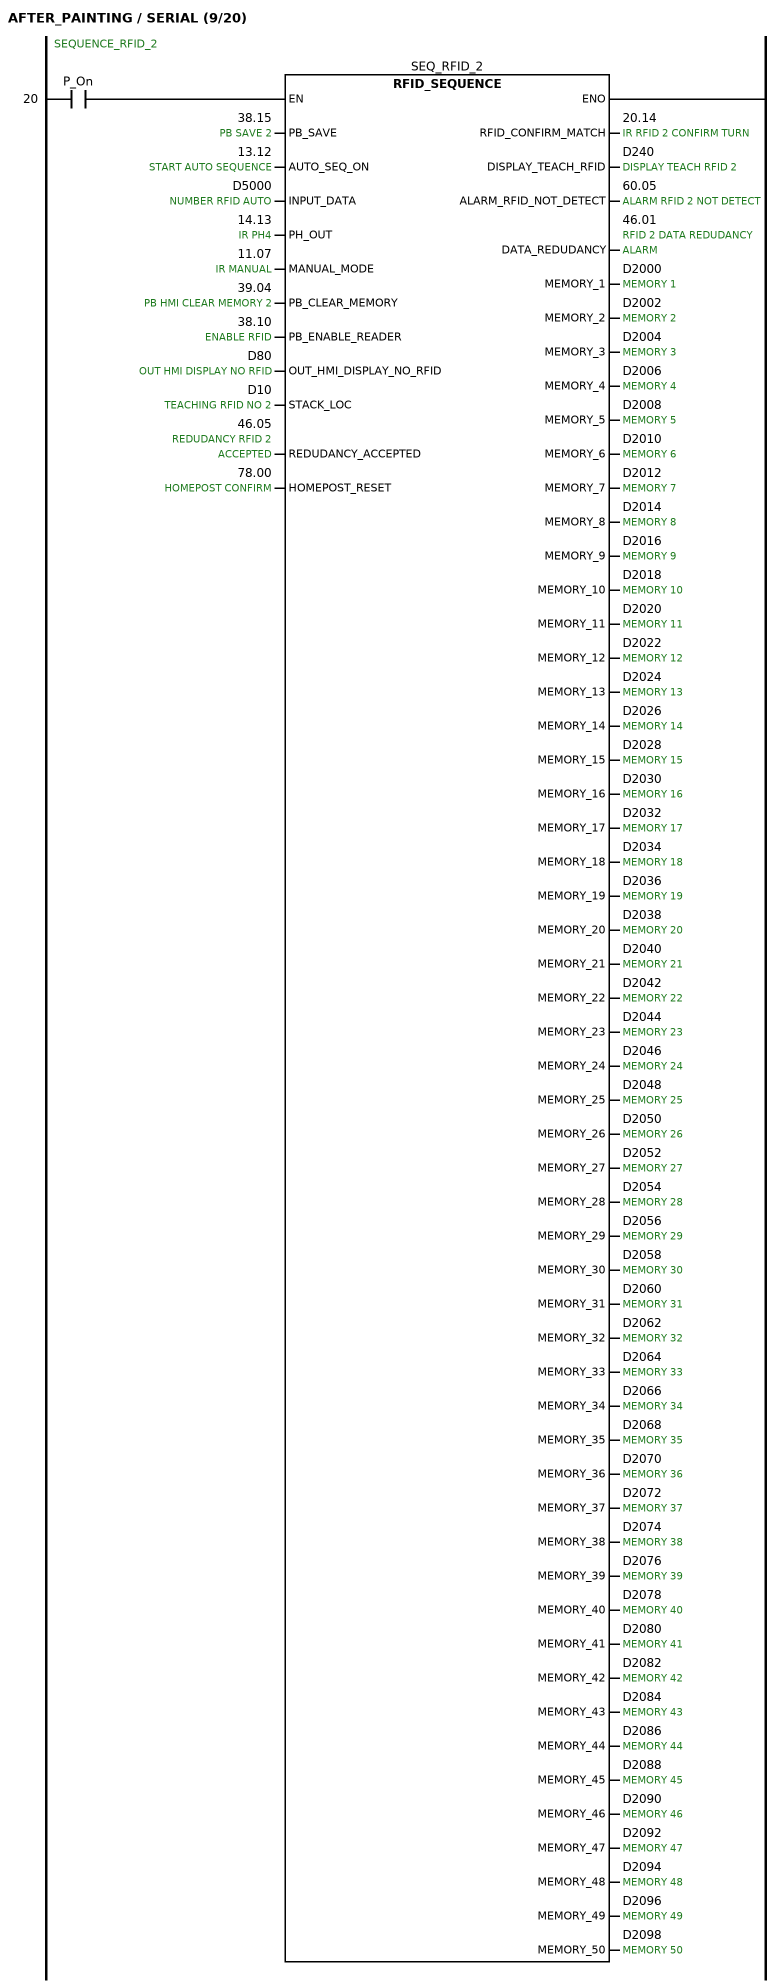
; [picture p72: AFTER_PAINTING / SERIAL, rungs 20-20]
; rung 20: SEQUENCE_RFID_2
LD P_On
CALL SEQ_RFID_2 : RFID_SEQUENCE (PB_SAVE := 38.15, AUTO_SEQ_ON := 13.12, INPUT_DATA := D5000, PH_OUT := 14.13, MANUAL_MODE := 11.07, PB_CLEAR_MEMORY := 39.04, PB_ENABLE_READER := 38.10, OUT_HMI_DISPLAY_NO_RFID := D80, STACK_LOC := D10, REDUDANCY_ACCEPTED := 46.05, HOMEPOST_RESET := 78.00, RFID_CONFIRM_MATCH => 20.14, DISPLAY_TEACH_RFID => D240, ALARM_RFID_NOT_DETECT => 60.05, DATA_REDUDANCY => 46.01, MEMORY_1 => D2000, MEMORY_2 => D2002, MEMORY_3 => D2004, MEMORY_4 => D2006, MEMORY_5 => D2008, MEMORY_6 => D2010, MEMORY_7 => D2012, MEMORY_8 => D2014, MEMORY_9 => D2016, MEMORY_10 => D2018, MEMORY_11 => D2020, MEMORY_12 => D2022, MEMORY_13 => D2024, MEMORY_14 => D2026, MEMORY_15 => D2028, MEMORY_16 => D2030, MEMORY_17 => D2032, MEMORY_18 => D2034, MEMORY_19 => D2036, MEMORY_20 => D2038, MEMORY_21 => D2040, MEMORY_22 => D2042, MEMORY_23 => D2044, MEMORY_24 => D2046, MEMORY_25 => D2048, MEMORY_26 => D2050, MEMORY_27 => D2052, MEMORY_28 => D2054, MEMORY_29 => D2056, MEMORY_30 => D2058, MEMORY_31 => D2060, MEMORY_32 => D2062, MEMORY_33 => D2064, MEMORY_34 => D2066, MEMORY_35 => D2068, MEMORY_36 => D2070, MEMORY_37 => D2072, MEMORY_38 => D2074, MEMORY_39 => D2076, MEMORY_40 => D2078, MEMORY_41 => D2080, MEMORY_42 => D2082, MEMORY_43 => D2084, MEMORY_44 => D2086, MEMORY_45 => D2088, MEMORY_46 => D2090, MEMORY_47 => D2092, MEMORY_48 => D2094, MEMORY_49 => D2096, MEMORY_50 => D2098)  ; PB SAVE 2, START AUTO SEQUENCE, NUMBER RFID AUTO, IR PH4, IR MANUAL, PB HMI CLEAR MEMORY 2, ENABLE RFID, OUT HMI DISPLAY NO RFID, TEACHING RFID NO 2, REDUDANCY RFID 2 ACCEPTED, HOMEPOST CONFIRM, IR RFID 2 CONFIRM TURN, DISPLAY TEACH RFID 2, ALARM RFID 2 NOT DETECT, RFID 2 DATA REDUDANCY ALARM, MEMORY 1, MEMORY 2, MEMORY 3, MEMORY 4, MEMORY 5, MEMORY 6, MEMORY 7, MEMORY 8, MEMORY 9, MEMORY 10, MEMORY 11, MEMORY 12, MEMORY 13, MEMORY 14, MEMORY 15, MEMORY 16, MEMORY 17, MEMORY 18, MEMORY 19, MEMORY 20, MEMORY 21, MEMORY 22, MEMORY 23, MEMORY 24, MEMORY 25, MEMORY 26, MEMORY 27, MEMORY 28, MEMORY 29, MEMORY 30, MEMORY 31, MEMORY 32, MEMORY 33, MEMORY 34, MEMORY 35, MEMORY 36, MEMORY 37, MEMORY 38, MEMORY 39, MEMORY 40, MEMORY 41, MEMORY 42, MEMORY 43, MEMORY 44, MEMORY 45, MEMORY 46, MEMORY 47, MEMORY 48, MEMORY 49, MEMORY 50

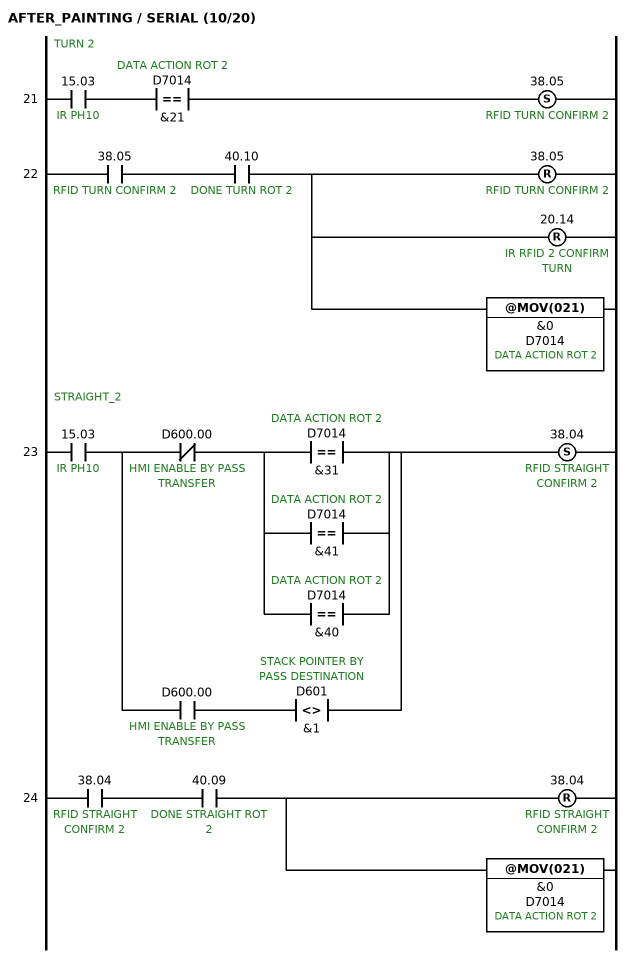
; rung 21: TURN 2
LD 15.03  ; IR PH10
AND=(300) D7014 &21  ; DATA ACTION ROT 2
SET 38.05  ; RFID TURN CONFIRM 2
; rung 22
LD 38.05  ; RFID TURN CONFIRM 2
AND 40.10  ; DONE TURN ROT 2
RSET 38.05  ; RFID TURN CONFIRM 2
RSET 20.14  ; IR RFID 2 CONFIRM TURN
@MOV(021) &0 D7014  ; DATA ACTION ROT 2
; rung 23: STRAIGHT_2
LD 15.03  ; IR PH10
LDNOT D600.00  ; HMI ENABLE BY PASS TRANSFER
LD=(300) D7014 &31  ; DATA ACTION ROT 2
OR=(300) D7014 &41  ; DATA ACTION ROT 2
OR=(300) D7014 &40  ; DATA ACTION ROT 2
ANDLD
LD D600.00  ; HMI ENABLE BY PASS TRANSFER
AND<>(305) D601 &1  ; STACK POINTER BY PASS DESTINATION
ORLD
ANDLD
SET 38.04  ; RFID STRAIGHT CONFIRM 2
; rung 24
LD 38.04  ; RFID STRAIGHT CONFIRM 2
AND 40.09  ; DONE STRAIGHT ROT 2
RSET 38.04  ; RFID STRAIGHT CONFIRM 2
@MOV(021) &0 D7014  ; DATA ACTION ROT 2

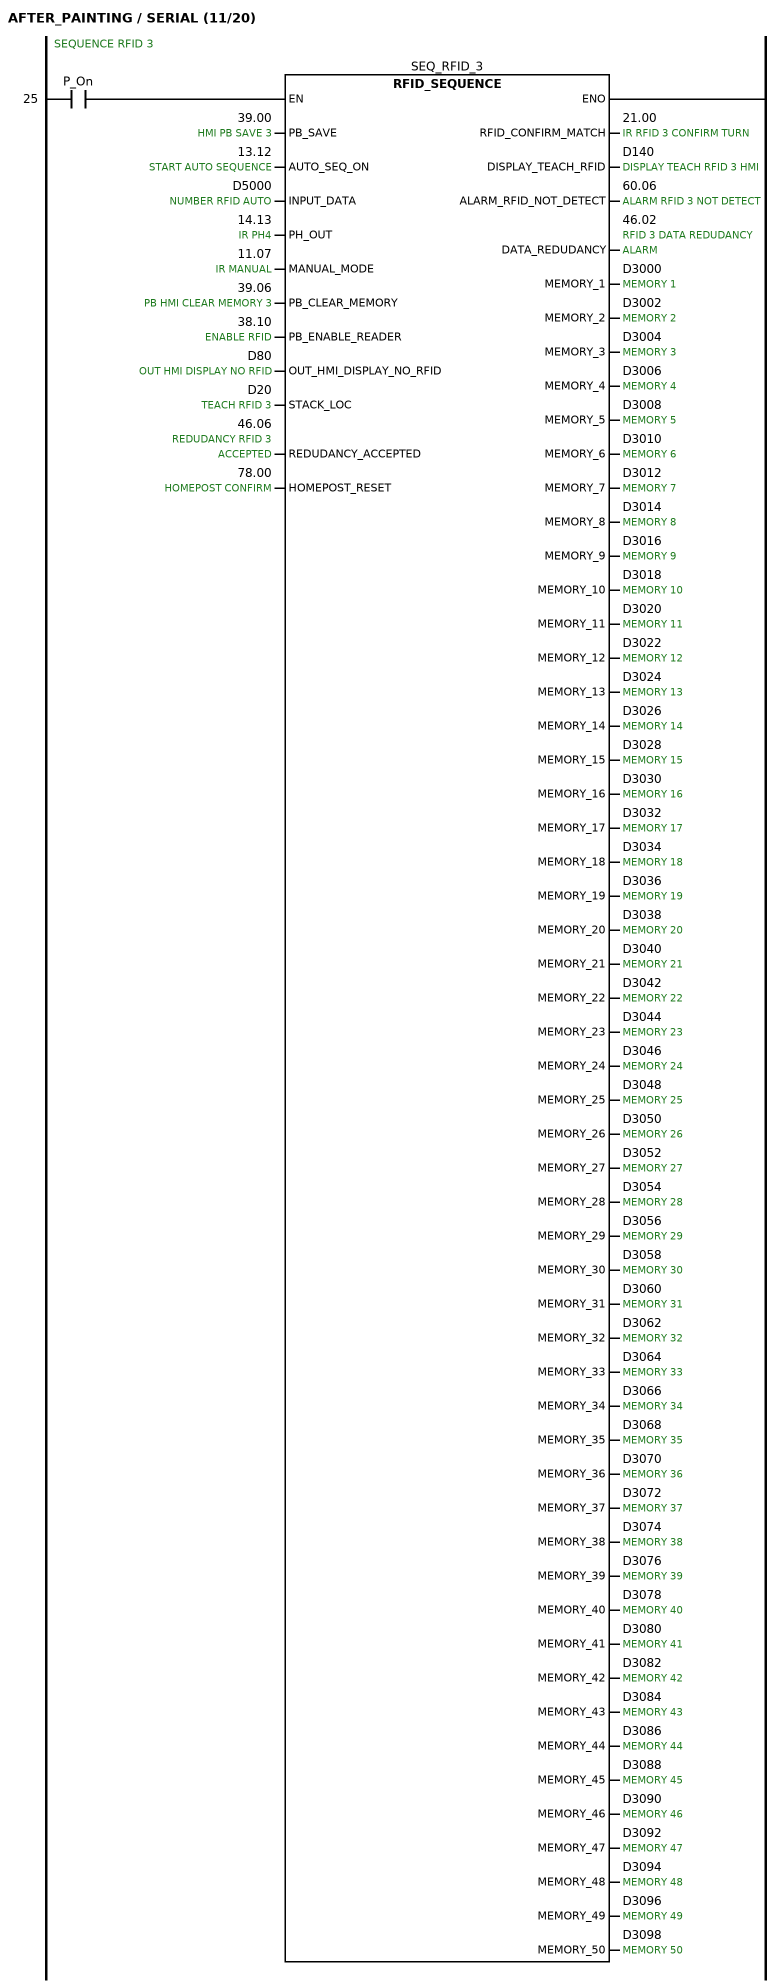
; rung 25: SEQUENCE RFID 3
LD P_On
CALL SEQ_RFID_3 : RFID_SEQUENCE (PB_SAVE := 39.00, AUTO_SEQ_ON := 13.12, INPUT_DATA := D5000, PH_OUT := 14.13, MANUAL_MODE := 11.07, PB_CLEAR_MEMORY := 39.06, PB_ENABLE_READER := 38.10, OUT_HMI_DISPLAY_NO_RFID := D80, STACK_LOC := D20, REDUDANCY_ACCEPTED := 46.06, HOMEPOST_RESET := 78.00, RFID_CONFIRM_MATCH => 21.00, DISPLAY_TEACH_RFID => D140, ALARM_RFID_NOT_DETECT => 60.06, DATA_REDUDANCY => 46.02, MEMORY_1 => D3000, MEMORY_2 => D3002, MEMORY_3 => D3004, MEMORY_4 => D3006, MEMORY_5 => D3008, MEMORY_6 => D3010, MEMORY_7 => D3012, MEMORY_8 => D3014, MEMORY_9 => D3016, MEMORY_10 => D3018, MEMORY_11 => D3020, MEMORY_12 => D3022, MEMORY_13 => D3024, MEMORY_14 => D3026, MEMORY_15 => D3028, MEMORY_16 => D3030, MEMORY_17 => D3032, MEMORY_18 => D3034, MEMORY_19 => D3036, MEMORY_20 => D3038, MEMORY_21 => D3040, MEMORY_22 => D3042, MEMORY_23 => D3044, MEMORY_24 => D3046, MEMORY_25 => D3048, MEMORY_26 => D3050, MEMORY_27 => D3052, MEMORY_28 => D3054, MEMORY_29 => D3056, MEMORY_30 => D3058, MEMORY_31 => D3060, MEMORY_32 => D3062, MEMORY_33 => D3064, MEMORY_34 => D3066, MEMORY_35 => D3068, MEMORY_36 => D3070, MEMORY_37 => D3072, MEMORY_38 => D3074, MEMORY_39 => D3076, MEMORY_40 => D3078, MEMORY_41 => D3080, MEMORY_42 => D3082, MEMORY_43 => D3084, MEMORY_44 => D3086, MEMORY_45 => D3088, MEMORY_46 => D3090, MEMORY_47 => D3092, MEMORY_48 => D3094, MEMORY_49 => D3096, MEMORY_50 => D3098)  ; HMI PB SAVE 3, START AUTO SEQUENCE, NUMBER RFID AUTO, IR PH4, IR MANUAL, PB HMI CLEAR MEMORY 3, ENABLE RFID, OUT HMI DISPLAY NO RFID, TEACH RFID 3, REDUDANCY RFID 3 ACCEPTED, HOMEPOST CONFIRM, IR RFID 3 CONFIRM TURN, DISPLAY TEACH RFID 3 HMI, ALARM RFID 3 NOT DETECT, RFID 3 DATA REDUDANCY ALARM, MEMORY 1, MEMORY 2, MEMORY 3, MEMORY 4, MEMORY 5, MEMORY 6, MEMORY 7, MEMORY 8, MEMORY 9, MEMORY 10, MEMORY 11, MEMORY 12, MEMORY 13, MEMORY 14, MEMORY 15, MEMORY 16, MEMORY 17, MEMORY 18, MEMORY 19, MEMORY 20, MEMORY 21, MEMORY 22, MEMORY 23, MEMORY 24, MEMORY 25, MEMORY 26, MEMORY 27, MEMORY 28, MEMORY 29, MEMORY 30, MEMORY 31, MEMORY 32, MEMORY 33, MEMORY 34, MEMORY 35, MEMORY 36, MEMORY 37, MEMORY 38, MEMORY 39, MEMORY 40, MEMORY 41, MEMORY 42, MEMORY 43, MEMORY 44, MEMORY 45, MEMORY 46, MEMORY 47, MEMORY 48, MEMORY 49, MEMORY 50

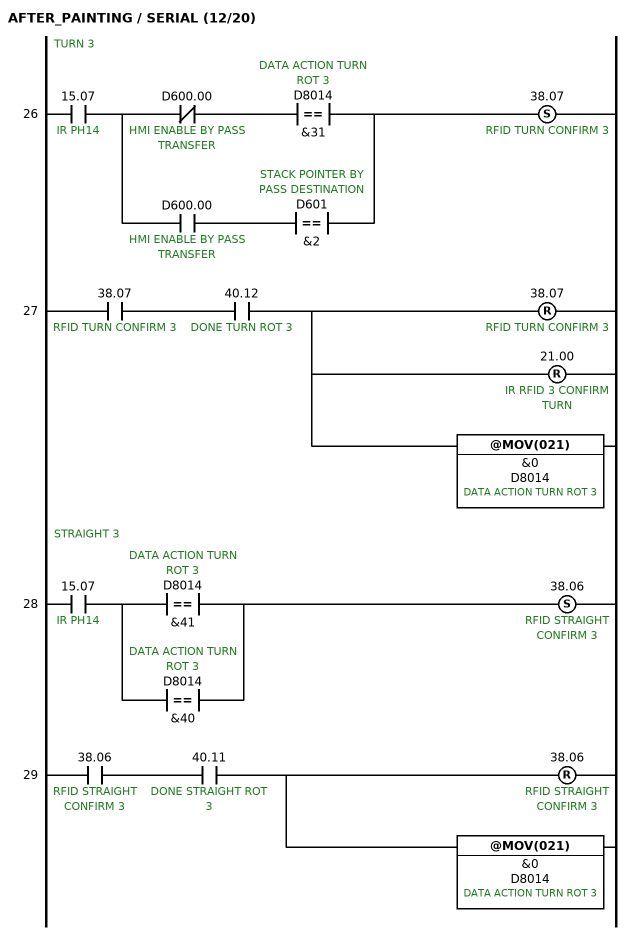
; rung 26: TURN 3
LD 15.07  ; IR PH14
LDNOT D600.00  ; HMI ENABLE BY PASS TRANSFER
AND=(300) D8014 &31  ; DATA ACTION TURN ROT 3
LD D600.00  ; HMI ENABLE BY PASS TRANSFER
AND=(300) D601 &2  ; STACK POINTER BY PASS DESTINATION
ORLD
ANDLD
SET 38.07  ; RFID TURN CONFIRM 3
; rung 27
LD 38.07  ; RFID TURN CONFIRM 3
AND 40.12  ; DONE TURN ROT 3
RSET 38.07  ; RFID TURN CONFIRM 3
RSET 21.00  ; IR RFID 3 CONFIRM TURN
@MOV(021) &0 D8014  ; DATA ACTION TURN ROT 3
; rung 28: STRAIGHT 3
LD 15.07  ; IR PH14
LD=(300) D8014 &41  ; DATA ACTION TURN ROT 3
OR=(300) D8014 &40  ; DATA ACTION TURN ROT 3
ANDLD
SET 38.06  ; RFID STRAIGHT CONFIRM 3
; rung 29
LD 38.06  ; RFID STRAIGHT CONFIRM 3
AND 40.11  ; DONE STRAIGHT ROT 3
RSET 38.06  ; RFID STRAIGHT CONFIRM 3
@MOV(021) &0 D8014  ; DATA ACTION TURN ROT 3

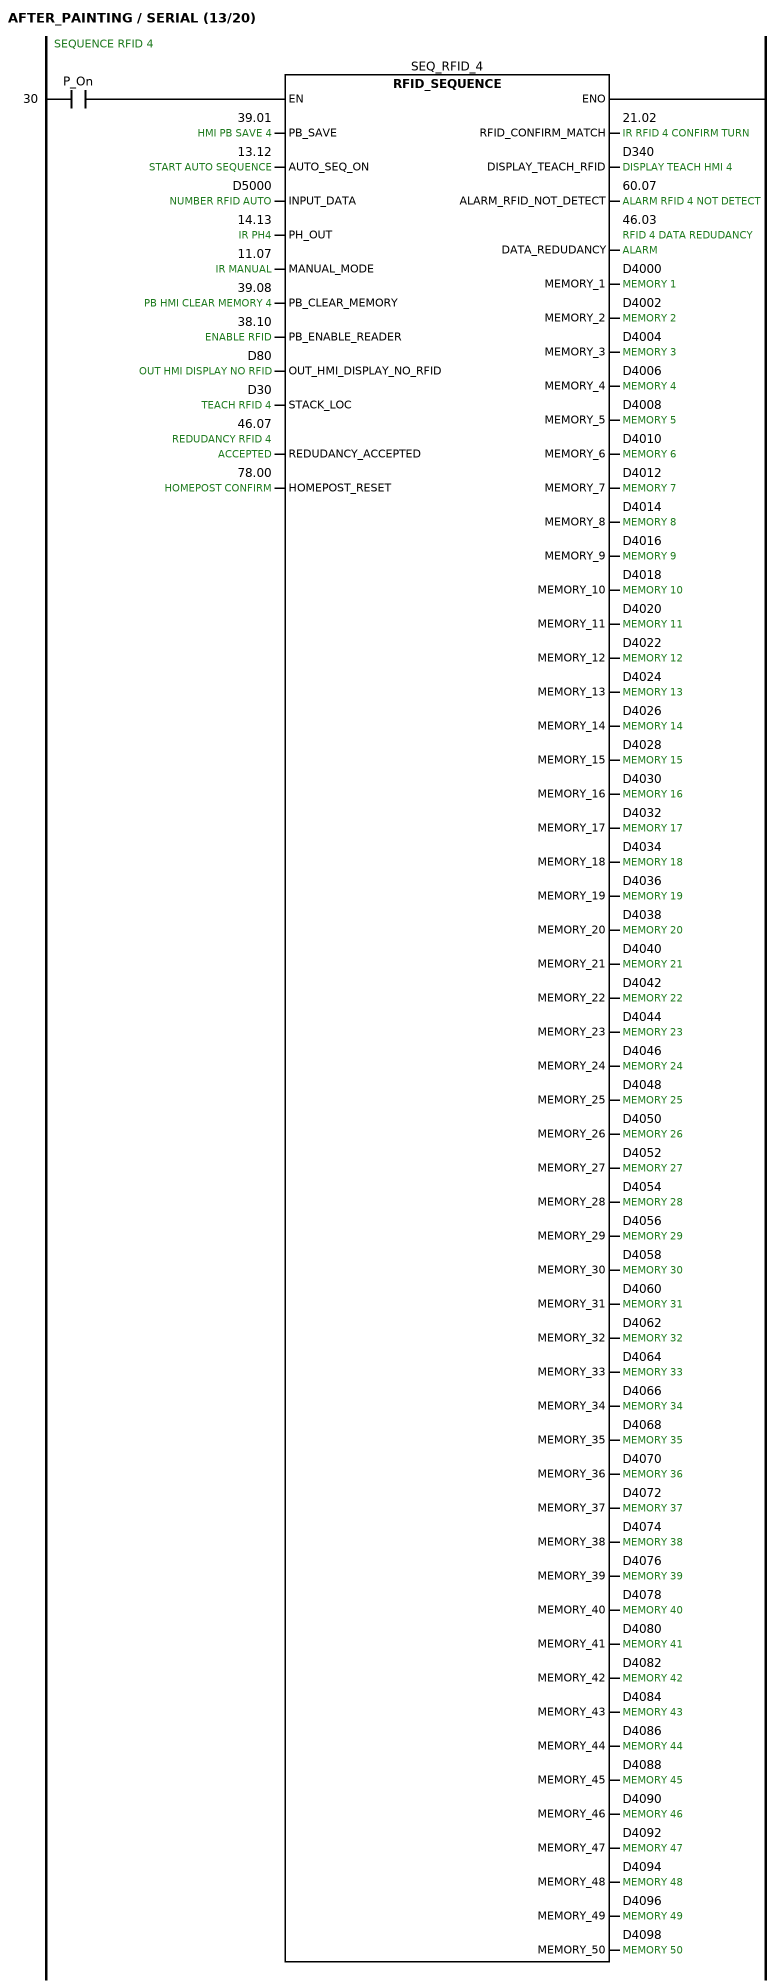
; rung 30: SEQUENCE RFID 4
LD P_On
CALL SEQ_RFID_4 : RFID_SEQUENCE (PB_SAVE := 39.01, AUTO_SEQ_ON := 13.12, INPUT_DATA := D5000, PH_OUT := 14.13, MANUAL_MODE := 11.07, PB_CLEAR_MEMORY := 39.08, PB_ENABLE_READER := 38.10, OUT_HMI_DISPLAY_NO_RFID := D80, STACK_LOC := D30, REDUDANCY_ACCEPTED := 46.07, HOMEPOST_RESET := 78.00, RFID_CONFIRM_MATCH => 21.02, DISPLAY_TEACH_RFID => D340, ALARM_RFID_NOT_DETECT => 60.07, DATA_REDUDANCY => 46.03, MEMORY_1 => D4000, MEMORY_2 => D4002, MEMORY_3 => D4004, MEMORY_4 => D4006, MEMORY_5 => D4008, MEMORY_6 => D4010, MEMORY_7 => D4012, MEMORY_8 => D4014, MEMORY_9 => D4016, MEMORY_10 => D4018, MEMORY_11 => D4020, MEMORY_12 => D4022, MEMORY_13 => D4024, MEMORY_14 => D4026, MEMORY_15 => D4028, MEMORY_16 => D4030, MEMORY_17 => D4032, MEMORY_18 => D4034, MEMORY_19 => D4036, MEMORY_20 => D4038, MEMORY_21 => D4040, MEMORY_22 => D4042, MEMORY_23 => D4044, MEMORY_24 => D4046, MEMORY_25 => D4048, MEMORY_26 => D4050, MEMORY_27 => D4052, MEMORY_28 => D4054, MEMORY_29 => D4056, MEMORY_30 => D4058, MEMORY_31 => D4060, MEMORY_32 => D4062, MEMORY_33 => D4064, MEMORY_34 => D4066, MEMORY_35 => D4068, MEMORY_36 => D4070, MEMORY_37 => D4072, MEMORY_38 => D4074, MEMORY_39 => D4076, MEMORY_40 => D4078, MEMORY_41 => D4080, MEMORY_42 => D4082, MEMORY_43 => D4084, MEMORY_44 => D4086, MEMORY_45 => D4088, MEMORY_46 => D4090, MEMORY_47 => D4092, MEMORY_48 => D4094, MEMORY_49 => D4096, MEMORY_50 => D4098)  ; HMI PB SAVE 4, START AUTO SEQUENCE, NUMBER RFID AUTO, IR PH4, IR MANUAL, PB HMI CLEAR MEMORY 4, ENABLE RFID, OUT HMI DISPLAY NO RFID, TEACH RFID 4, REDUDANCY RFID 4 ACCEPTED, HOMEPOST CONFIRM, IR RFID 4 CONFIRM TURN, DISPLAY TEACH HMI 4, ALARM RFID 4 NOT DETECT, RFID 4 DATA REDUDANCY ALARM, MEMORY 1, MEMORY 2, MEMORY 3, MEMORY 4, MEMORY 5, MEMORY 6, MEMORY 7, MEMORY 8, MEMORY 9, MEMORY 10, MEMORY 11, MEMORY 12, MEMORY 13, MEMORY 14, MEMORY 15, MEMORY 16, MEMORY 17, MEMORY 18, MEMORY 19, MEMORY 20, MEMORY 21, MEMORY 22, MEMORY 23, MEMORY 24, MEMORY 25, MEMORY 26, MEMORY 27, MEMORY 28, MEMORY 29, MEMORY 30, MEMORY 31, MEMORY 32, MEMORY 33, MEMORY 34, MEMORY 35, MEMORY 36, MEMORY 37, MEMORY 38, MEMORY 39, MEMORY 40, MEMORY 41, MEMORY 42, MEMORY 43, MEMORY 44, MEMORY 45, MEMORY 46, MEMORY 47, MEMORY 48, MEMORY 49, MEMORY 50

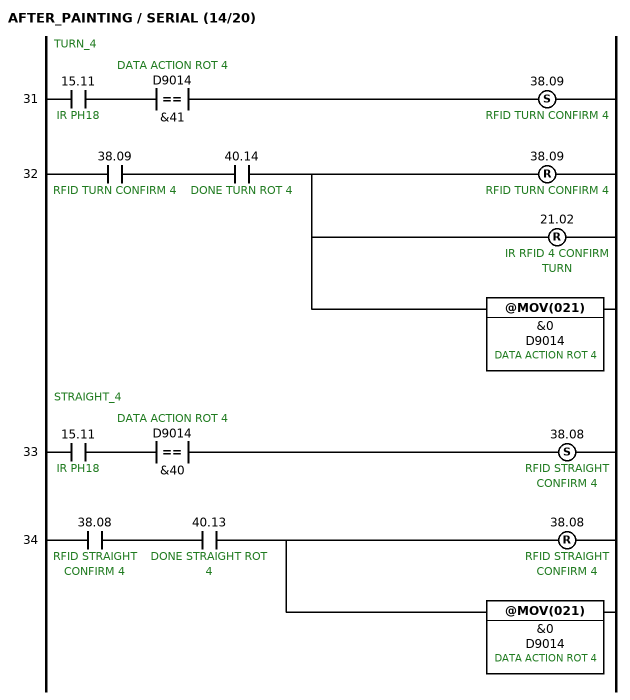
; rung 31: TURN_4
LD 15.11  ; IR PH18
AND=(300) D9014 &41  ; DATA ACTION ROT 4
SET 38.09  ; RFID TURN CONFIRM 4
; rung 32
LD 38.09  ; RFID TURN CONFIRM 4
AND 40.14  ; DONE TURN ROT 4
RSET 38.09  ; RFID TURN CONFIRM 4
RSET 21.02  ; IR RFID 4 CONFIRM TURN
@MOV(021) &0 D9014  ; DATA ACTION ROT 4
; rung 33: STRAIGHT_4
LD 15.11  ; IR PH18
AND=(300) D9014 &40  ; DATA ACTION ROT 4
SET 38.08  ; RFID STRAIGHT CONFIRM 4
; rung 34
LD 38.08  ; RFID STRAIGHT CONFIRM 4
AND 40.13  ; DONE STRAIGHT ROT 4
RSET 38.08  ; RFID STRAIGHT CONFIRM 4
@MOV(021) &0 D9014  ; DATA ACTION ROT 4

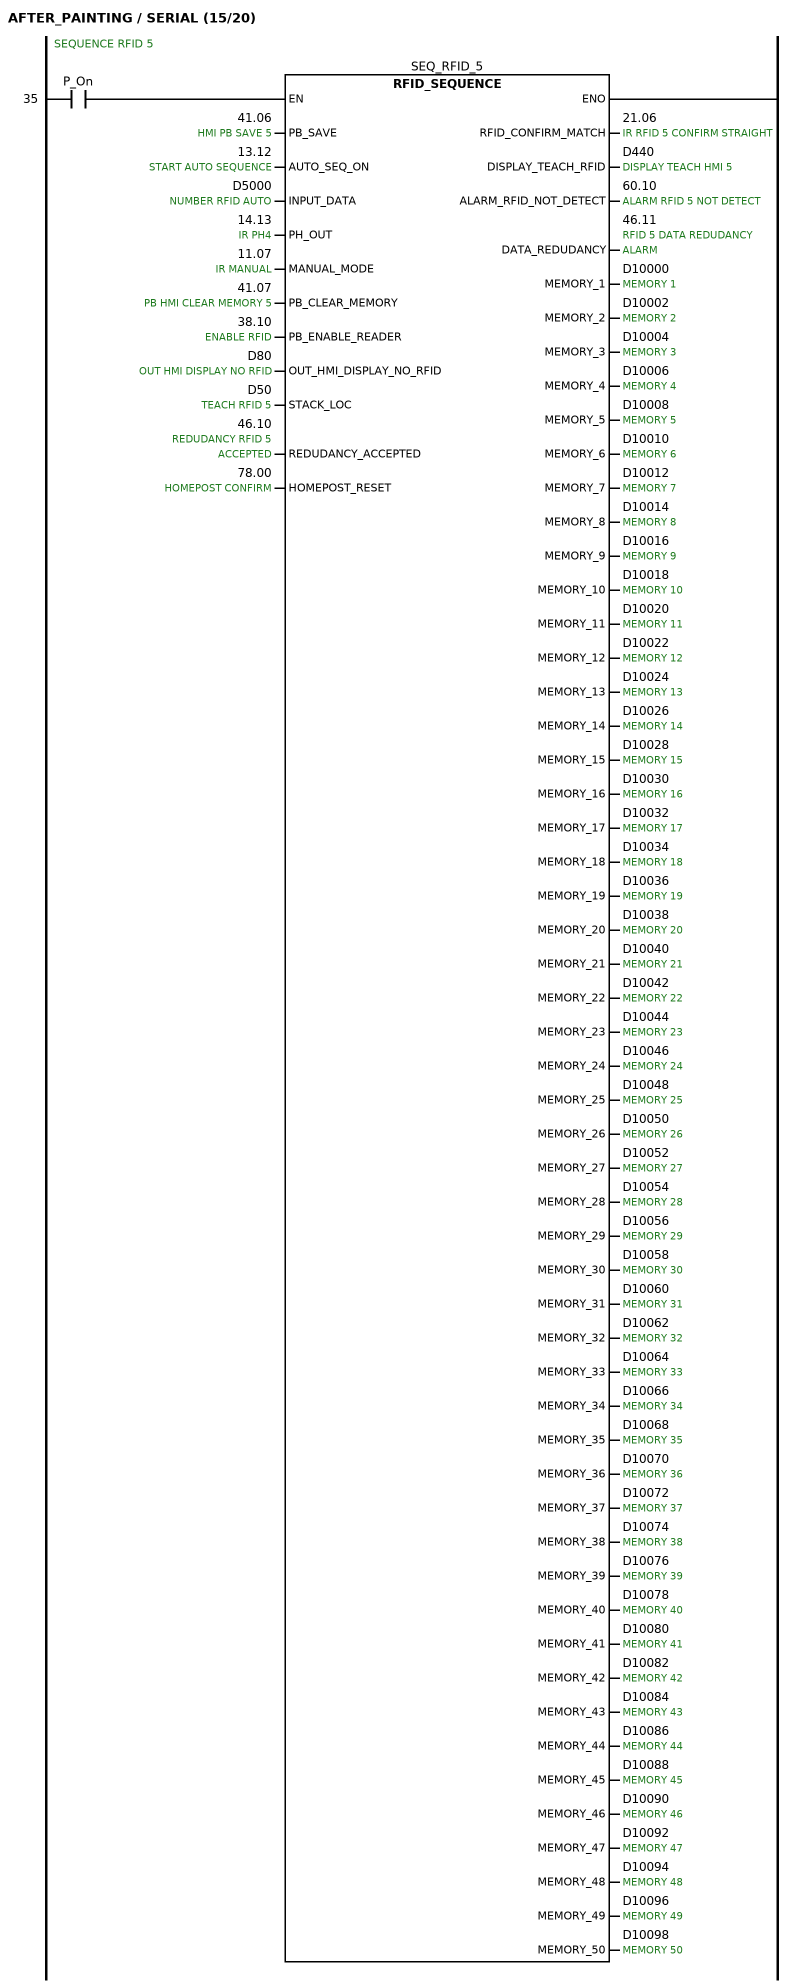
; rung 35: SEQUENCE RFID 5
LD P_On
CALL SEQ_RFID_5 : RFID_SEQUENCE (PB_SAVE := 41.06, AUTO_SEQ_ON := 13.12, INPUT_DATA := D5000, PH_OUT := 14.13, MANUAL_MODE := 11.07, PB_CLEAR_MEMORY := 41.07, PB_ENABLE_READER := 38.10, OUT_HMI_DISPLAY_NO_RFID := D80, STACK_LOC := D50, REDUDANCY_ACCEPTED := 46.10, HOMEPOST_RESET := 78.00, RFID_CONFIRM_MATCH => 21.06, DISPLAY_TEACH_RFID => D440, ALARM_RFID_NOT_DETECT => 60.10, DATA_REDUDANCY => 46.11, MEMORY_1 => D10000, MEMORY_2 => D10002, MEMORY_3 => D10004, MEMORY_4 => D10006, MEMORY_5 => D10008, MEMORY_6 => D10010, MEMORY_7 => D10012, MEMORY_8 => D10014, MEMORY_9 => D10016, MEMORY_10 => D10018, MEMORY_11 => D10020, MEMORY_12 => D10022, MEMORY_13 => D10024, MEMORY_14 => D10026, MEMORY_15 => D10028, MEMORY_16 => D10030, MEMORY_17 => D10032, MEMORY_18 => D10034, MEMORY_19 => D10036, MEMORY_20 => D10038, MEMORY_21 => D10040, MEMORY_22 => D10042, MEMORY_23 => D10044, MEMORY_24 => D10046, MEMORY_25 => D10048, MEMORY_26 => D10050, MEMORY_27 => D10052, MEMORY_28 => D10054, MEMORY_29 => D10056, MEMORY_30 => D10058, MEMORY_31 => D10060, MEMORY_32 => D10062, MEMORY_33 => D10064, MEMORY_34 => D10066, MEMORY_35 => D10068, MEMORY_36 => D10070, MEMORY_37 => D10072, MEMORY_38 => D10074, MEMORY_39 => D10076, MEMORY_40 => D10078, MEMORY_41 => D10080, MEMORY_42 => D10082, MEMORY_43 => D10084, MEMORY_44 => D10086, MEMORY_45 => D10088, MEMORY_46 => D10090, MEMORY_47 => D10092, MEMORY_48 => D10094, MEMORY_49 => D10096, MEMORY_50 => D10098)  ; HMI PB SAVE 5, START AUTO SEQUENCE, NUMBER RFID AUTO, IR PH4, IR MANUAL, PB HMI CLEAR MEMORY 5, ENABLE RFID, OUT HMI DISPLAY NO RFID, TEACH RFID 5, REDUDANCY RFID 5 ACCEPTED, HOMEPOST CONFIRM, IR RFID 5 CONFIRM STRAIGHT, DISPLAY TEACH HMI 5, ALARM RFID 5 NOT DETECT, RFID 5 DATA REDUDANCY ALARM, MEMORY 1, MEMORY 2, MEMORY 3, MEMORY 4, MEMORY 5, MEMORY 6, MEMORY 7, MEMORY 8, MEMORY 9, MEMORY 10, MEMORY 11, MEMORY 12, MEMORY 13, MEMORY 14, MEMORY 15, MEMORY 16, MEMORY 17, MEMORY 18, MEMORY 19, MEMORY 20, MEMORY 21, MEMORY 22, MEMORY 23, MEMORY 24, MEMORY 25, MEMORY 26, MEMORY 27, MEMORY 28, MEMORY 29, MEMORY 30, MEMORY 31, MEMORY 32, MEMORY 33, MEMORY 34, MEMORY 35, MEMORY 36, MEMORY 37, MEMORY 38, MEMORY 39, MEMORY 40, MEMORY 41, MEMORY 42, MEMORY 43, MEMORY 44, MEMORY 45, MEMORY 46, MEMORY 47, MEMORY 48, MEMORY 49, MEMORY 50

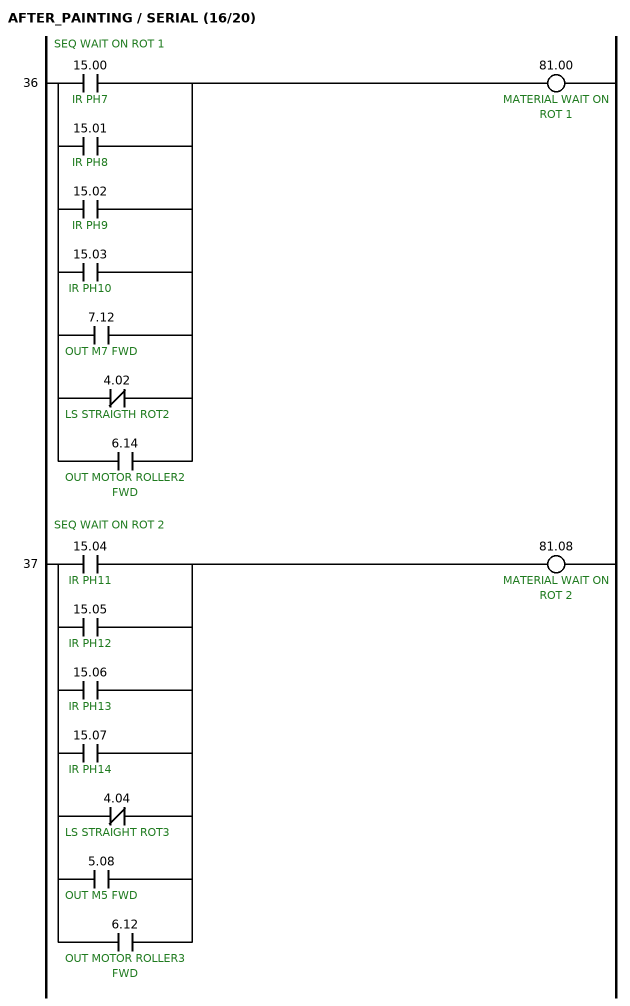
; rung 36: SEQ WAIT ON ROT 1
LD 15.00  ; IR PH7
OR 15.01  ; IR PH8
OR 15.02  ; IR PH9
OR 15.03  ; IR PH10
OR 7.12  ; OUT M7 FWD
ORNOT 4.02  ; LS STRAIGTH ROT2
OR 6.14  ; OUT MOTOR ROLLER2 FWD
OUT 81.00  ; MATERIAL WAIT ON ROT 1
; rung 37: SEQ WAIT ON ROT 2
LD 15.04  ; IR PH11
OR 15.05  ; IR PH12
OR 15.06  ; IR PH13
OR 15.07  ; IR PH14
ORNOT 4.04  ; LS STRAIGHT ROT3
OR 5.08  ; OUT M5 FWD
OR 6.12  ; OUT MOTOR ROLLER3 FWD
OUT 81.08  ; MATERIAL WAIT ON ROT 2

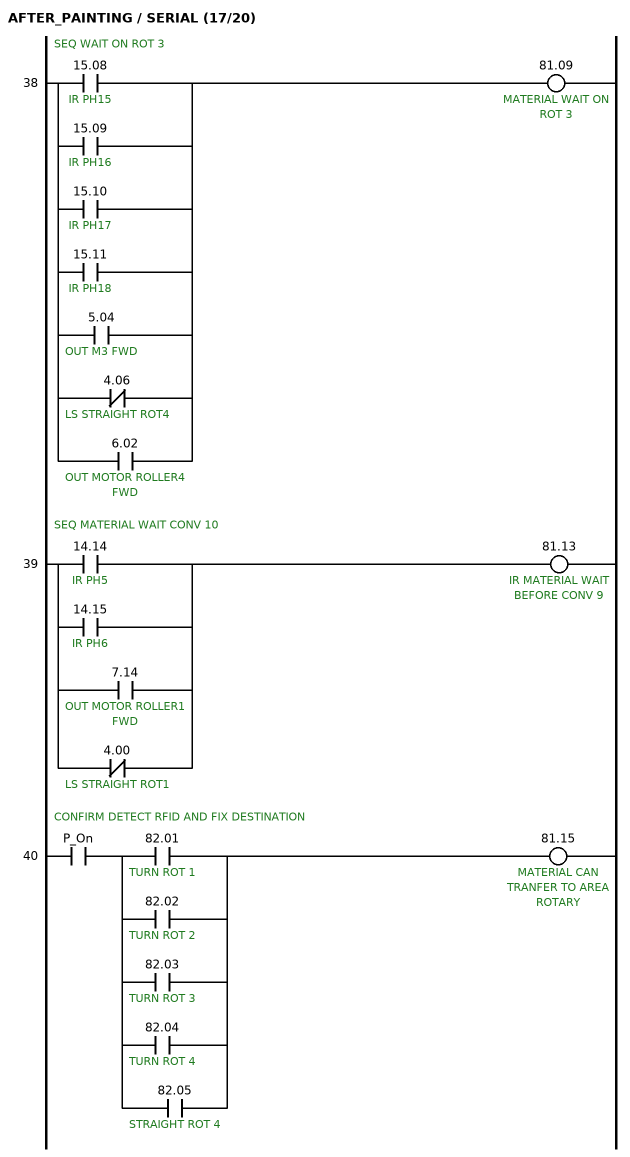
; rung 38: SEQ WAIT ON ROT 3
LD 15.08  ; IR PH15
OR 15.09  ; IR PH16
OR 15.10  ; IR PH17
OR 15.11  ; IR PH18
OR 5.04  ; OUT M3 FWD
ORNOT 4.06  ; LS STRAIGHT ROT4
OR 6.02  ; OUT MOTOR ROLLER4 FWD
OUT 81.09  ; MATERIAL WAIT ON ROT 3
; rung 39: SEQ MATERIAL WAIT CONV 10
LD 14.14  ; IR PH5
OR 14.15  ; IR PH6
OR 7.14  ; OUT MOTOR ROLLER1 FWD
ORNOT 4.00  ; LS STRAIGHT ROT1
OUT 81.13  ; IR MATERIAL WAIT BEFORE CONV 9
; rung 40: CONFIRM DETECT RFID AND FIX DESTINATION
LD P_On
LD 82.01  ; TURN ROT 1
OR 82.02  ; TURN ROT 2
OR 82.03  ; TURN ROT 3
OR 82.04  ; TURN ROT 4
OR 82.05  ; STRAIGHT ROT 4
ANDLD
OUT 81.15  ; MATERIAL CAN TRANFER TO AREA ROTARY

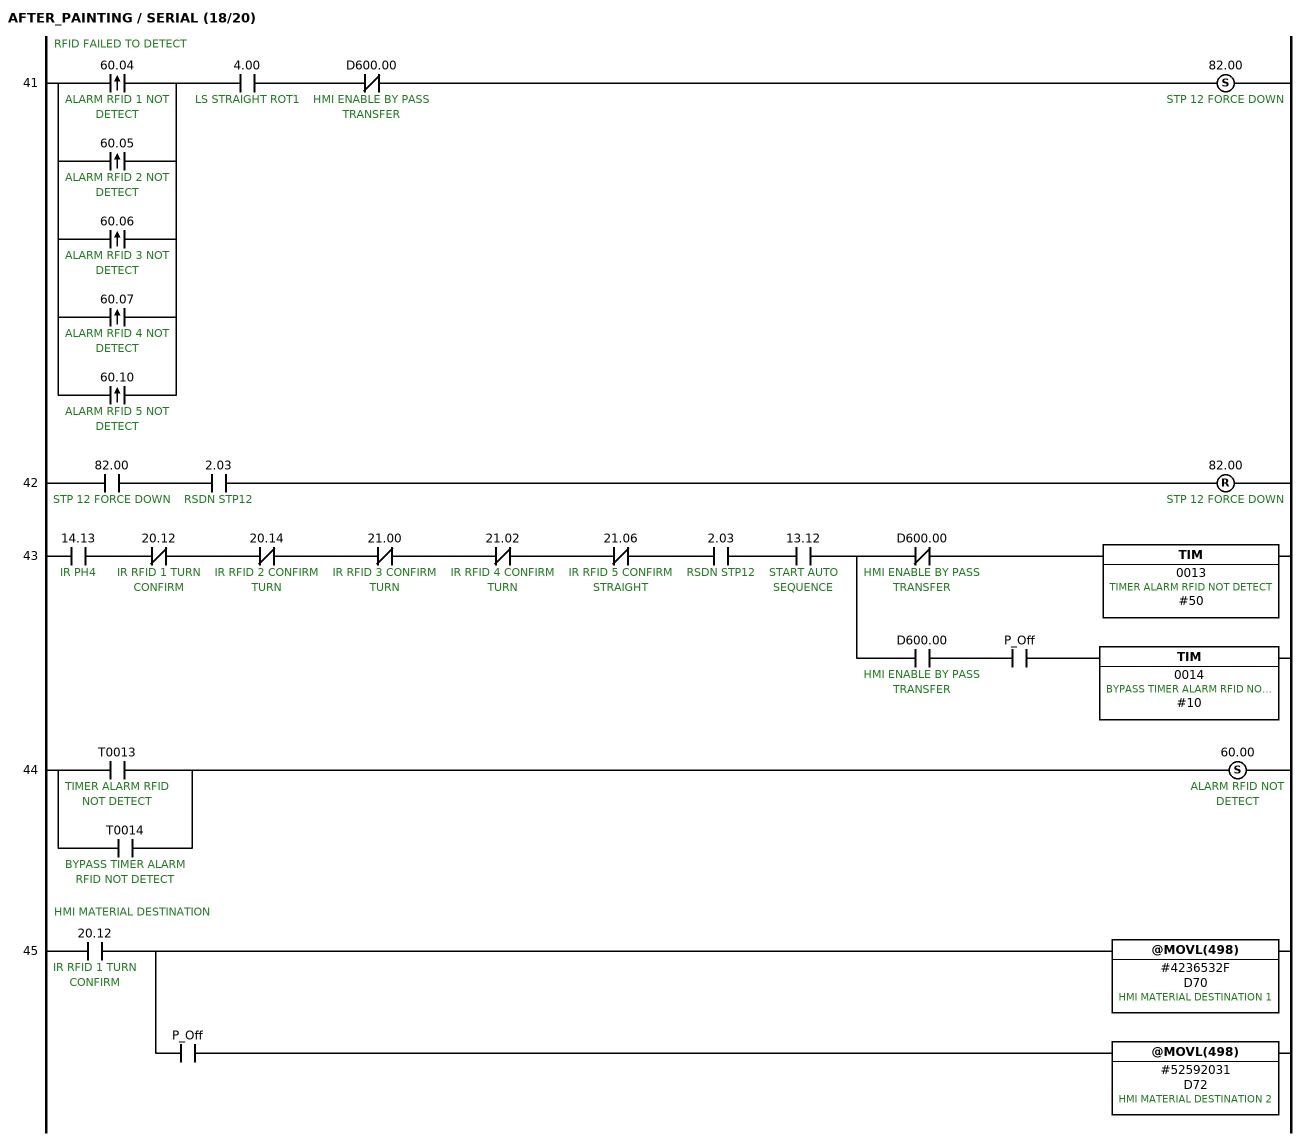
; rung 41: RFID FAILED TO DETECT
@LD 60.04  ; ALARM RFID 1 NOT DETECT
@OR 60.05  ; ALARM RFID 2 NOT DETECT
@OR 60.06  ; ALARM RFID 3 NOT DETECT
@OR 60.07  ; ALARM RFID 4 NOT DETECT
@OR 60.10  ; ALARM RFID 5 NOT DETECT
AND 4.00  ; LS STRAIGHT ROT1
ANDNOT D600.00  ; HMI ENABLE BY PASS TRANSFER
SET 82.00  ; STP 12 FORCE DOWN
; rung 42
LD 82.00  ; STP 12 FORCE DOWN
AND 2.03  ; RSDN STP12
RSET 82.00  ; STP 12 FORCE DOWN
; rung 43
LD 14.13  ; IR PH4
ANDNOT 20.12  ; IR RFID 1 TURN CONFIRM
ANDNOT 20.14  ; IR RFID 2 CONFIRM TURN
ANDNOT 21.00  ; IR RFID 3 CONFIRM TURN
ANDNOT 21.02  ; IR RFID 4 CONFIRM TURN
ANDNOT 21.06  ; IR RFID 5 CONFIRM STRAIGHT
AND 2.03  ; RSDN STP12
AND 13.12  ; START AUTO SEQUENCE
OUT TR0
ANDNOT D600.00  ; HMI ENABLE BY PASS TRANSFER
TIM 0013 #50  ; TIMER ALARM RFID NOT DETECT
LD TR0
AND D600.00  ; HMI ENABLE BY PASS TRANSFER
AND P_Off
TIM 0014 #10  ; BYPASS TIMER ALARM RFID NOT DETECT
; rung 44
LD T0013  ; TIMER ALARM RFID NOT DETECT
OR T0014  ; BYPASS TIMER ALARM RFID NOT DETECT
SET 60.00  ; ALARM RFID NOT DETECT
; rung 45: HMI MATERIAL DESTINATION
LD 20.12  ; IR RFID 1 TURN CONFIRM
@MOVL(498) #4236532F D70  ; HMI MATERIAL DESTINATION 1
AND P_Off
@MOVL(498) #52592031 D72  ; HMI MATERIAL DESTINATION 2

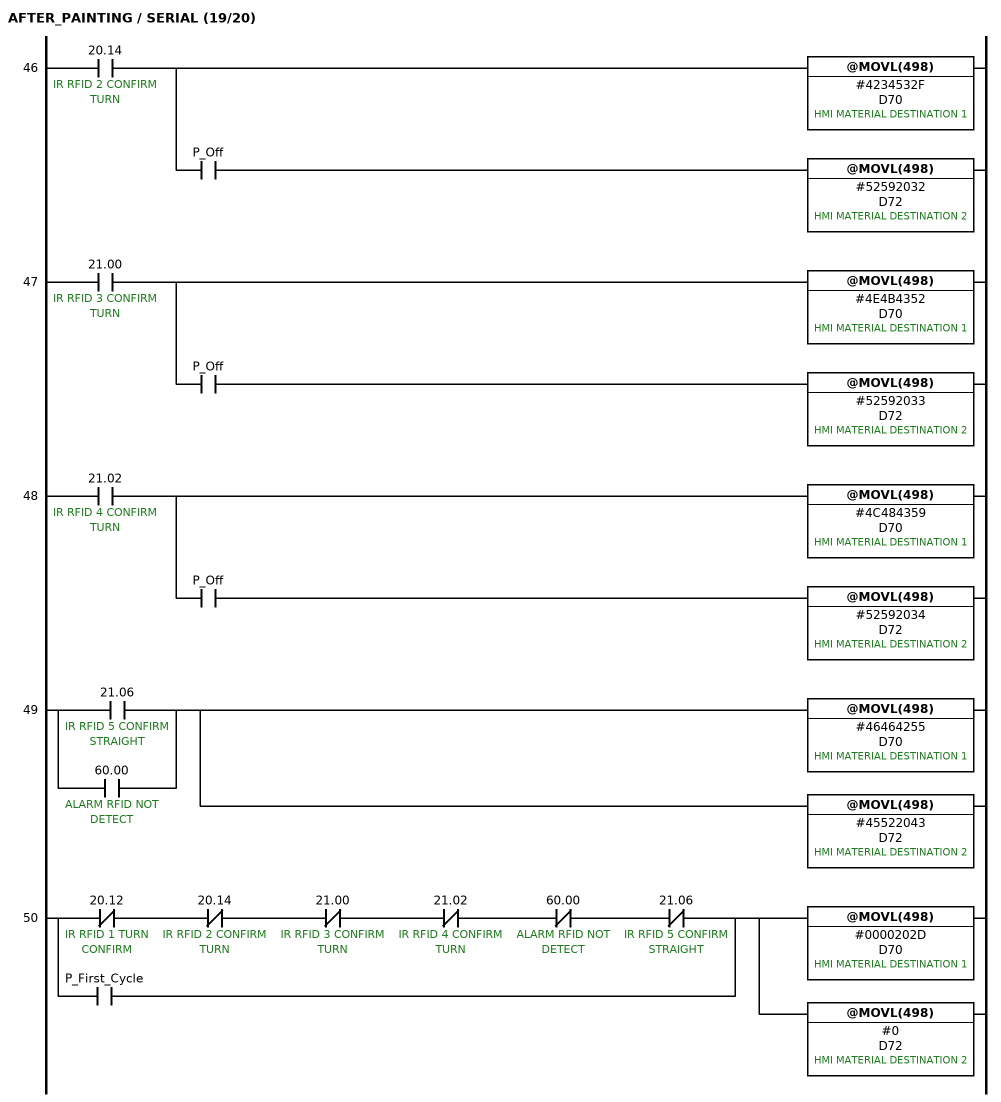
; rung 46
LD 20.14  ; IR RFID 2 CONFIRM TURN
@MOVL(498) #4234532F D70  ; HMI MATERIAL DESTINATION 1
AND P_Off
@MOVL(498) #52592032 D72  ; HMI MATERIAL DESTINATION 2
; rung 47
LD 21.00  ; IR RFID 3 CONFIRM TURN
@MOVL(498) #4E4B4352 D70  ; HMI MATERIAL DESTINATION 1
AND P_Off
@MOVL(498) #52592033 D72  ; HMI MATERIAL DESTINATION 2
; rung 48
LD 21.02  ; IR RFID 4 CONFIRM TURN
@MOVL(498) #4C484359 D70  ; HMI MATERIAL DESTINATION 1
AND P_Off
@MOVL(498) #52592034 D72  ; HMI MATERIAL DESTINATION 2
; rung 49
LD 21.06  ; IR RFID 5 CONFIRM STRAIGHT
OR 60.00  ; ALARM RFID NOT DETECT
@MOVL(498) #46464255 D70  ; HMI MATERIAL DESTINATION 1
@MOVL(498) #45522043 D72  ; HMI MATERIAL DESTINATION 2
; rung 50
LDNOT 20.12  ; IR RFID 1 TURN CONFIRM
ANDNOT 20.14  ; IR RFID 2 CONFIRM TURN
ANDNOT 21.00  ; IR RFID 3 CONFIRM TURN
ANDNOT 21.02  ; IR RFID 4 CONFIRM TURN
ANDNOT 60.00  ; ALARM RFID NOT DETECT
ANDNOT 21.06  ; IR RFID 5 CONFIRM STRAIGHT
OR P_First_Cycle
@MOVL(498) #0000202D D70  ; HMI MATERIAL DESTINATION 1
@MOVL(498) #0 D72  ; HMI MATERIAL DESTINATION 2

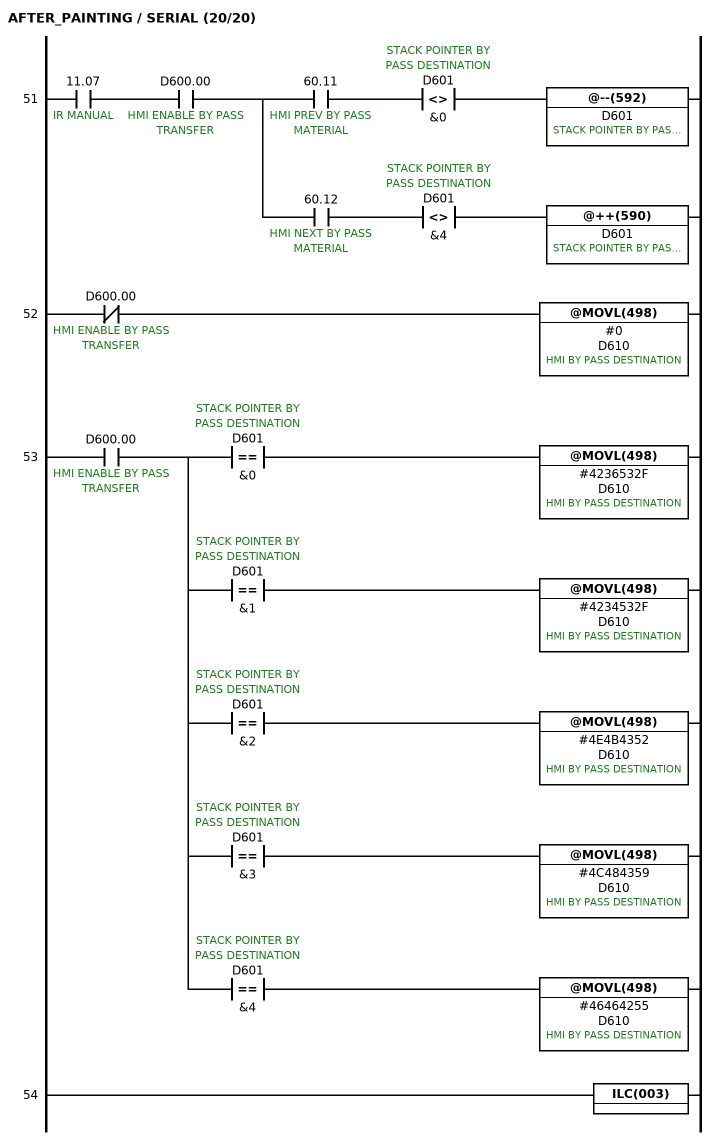
; rung 51
LD 11.07  ; IR MANUAL
AND D600.00  ; HMI ENABLE BY PASS TRANSFER
OUT TR0
AND 60.11  ; HMI PREV BY PASS MATERIAL
AND<>(305) D601 &0  ; STACK POINTER BY PASS DESTINATION
@--(592) D601  ; STACK POINTER BY PASS DESTINATION
LD TR0
AND 60.12  ; HMI NEXT BY PASS MATERIAL
AND<>(305) D601 &4  ; STACK POINTER BY PASS DESTINATION
@++(590) D601  ; STACK POINTER BY PASS DESTINATION
; rung 52
LDNOT D600.00  ; HMI ENABLE BY PASS TRANSFER
@MOVL(498) #0 D610  ; HMI BY PASS DESTINATION
; rung 53
LD D600.00  ; HMI ENABLE BY PASS TRANSFER
OUT TR0
AND=(300) D601 &0  ; STACK POINTER BY PASS DESTINATION
@MOVL(498) #4236532F D610  ; HMI BY PASS DESTINATION
LD TR0
AND=(300) D601 &1  ; STACK POINTER BY PASS DESTINATION
@MOVL(498) #4234532F D610  ; HMI BY PASS DESTINATION
LD TR0
AND=(300) D601 &2  ; STACK POINTER BY PASS DESTINATION
@MOVL(498) #4E4B4352 D610  ; HMI BY PASS DESTINATION
LD TR0
AND=(300) D601 &3  ; STACK POINTER BY PASS DESTINATION
@MOVL(498) #4C484359 D610  ; HMI BY PASS DESTINATION
LD TR0
AND=(300) D601 &4  ; STACK POINTER BY PASS DESTINATION
@MOVL(498) #46464255 D610  ; HMI BY PASS DESTINATION
; rung 54
ILC(003)

### Section WAIT_LIST

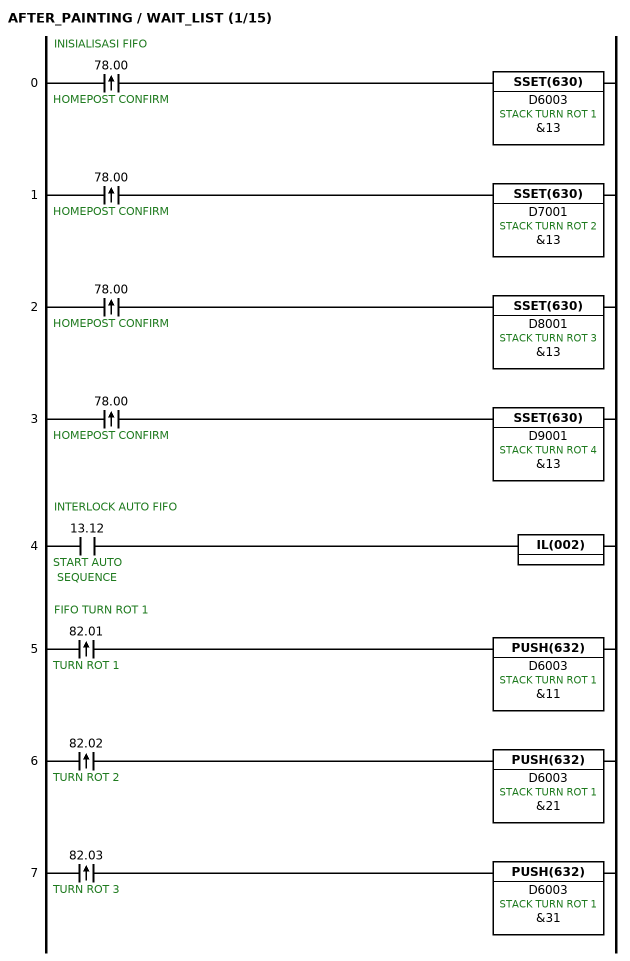
; rung 0: INISIALISASI FIFO
@LD 78.00  ; HOMEPOST CONFIRM
SSET(630) D6003 &13  ; STACK TURN ROT 1
; rung 1
@LD 78.00  ; HOMEPOST CONFIRM
SSET(630) D7001 &13  ; STACK TURN ROT 2
; rung 2
@LD 78.00  ; HOMEPOST CONFIRM
SSET(630) D8001 &13  ; STACK TURN ROT 3
; rung 3
@LD 78.00  ; HOMEPOST CONFIRM
SSET(630) D9001 &13  ; STACK TURN ROT 4
; rung 4: INTERLOCK AUTO FIFO
LD 13.12  ; START AUTO SEQUENCE
IL(002)
; rung 5: FIFO TURN ROT 1
@LD 82.01  ; TURN ROT 1
PUSH(632) D6003 &11  ; STACK TURN ROT 1
; rung 6
@LD 82.02  ; TURN ROT 2
PUSH(632) D6003 &21  ; STACK TURN ROT 1
; rung 7
@LD 82.03  ; TURN ROT 3
PUSH(632) D6003 &31  ; STACK TURN ROT 1

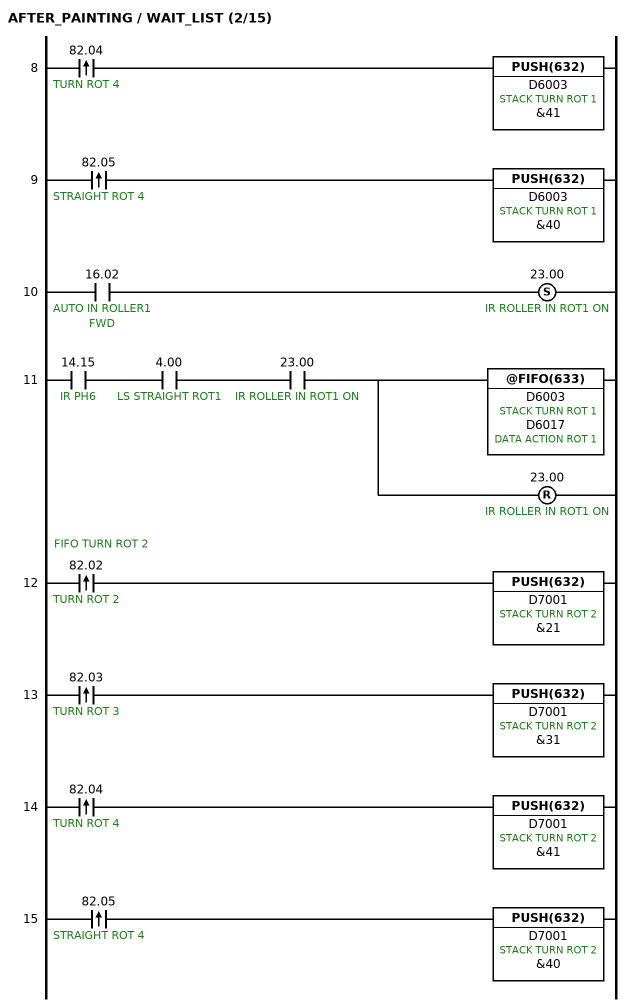
; rung 8
@LD 82.04  ; TURN ROT 4
PUSH(632) D6003 &41  ; STACK TURN ROT 1
; rung 9
@LD 82.05  ; STRAIGHT ROT 4
PUSH(632) D6003 &40  ; STACK TURN ROT 1
; rung 10
LD 16.02  ; AUTO IN ROLLER1 FWD
SET 23.00  ; IR ROLLER IN ROT1 ON
; rung 11
LD 14.15  ; IR PH6
AND 4.00  ; LS STRAIGHT ROT1
AND 23.00  ; IR ROLLER IN ROT1 ON
@FIFO(633) D6003 D6017  ; STACK TURN ROT 1, DATA ACTION ROT 1
RSET 23.00  ; IR ROLLER IN ROT1 ON
; rung 12: FIFO TURN ROT 2
@LD 82.02  ; TURN ROT 2
PUSH(632) D7001 &21  ; STACK TURN ROT 2
; rung 13
@LD 82.03  ; TURN ROT 3
PUSH(632) D7001 &31  ; STACK TURN ROT 2
; rung 14
@LD 82.04  ; TURN ROT 4
PUSH(632) D7001 &41  ; STACK TURN ROT 2
; rung 15
@LD 82.05  ; STRAIGHT ROT 4
PUSH(632) D7001 &40  ; STACK TURN ROT 2

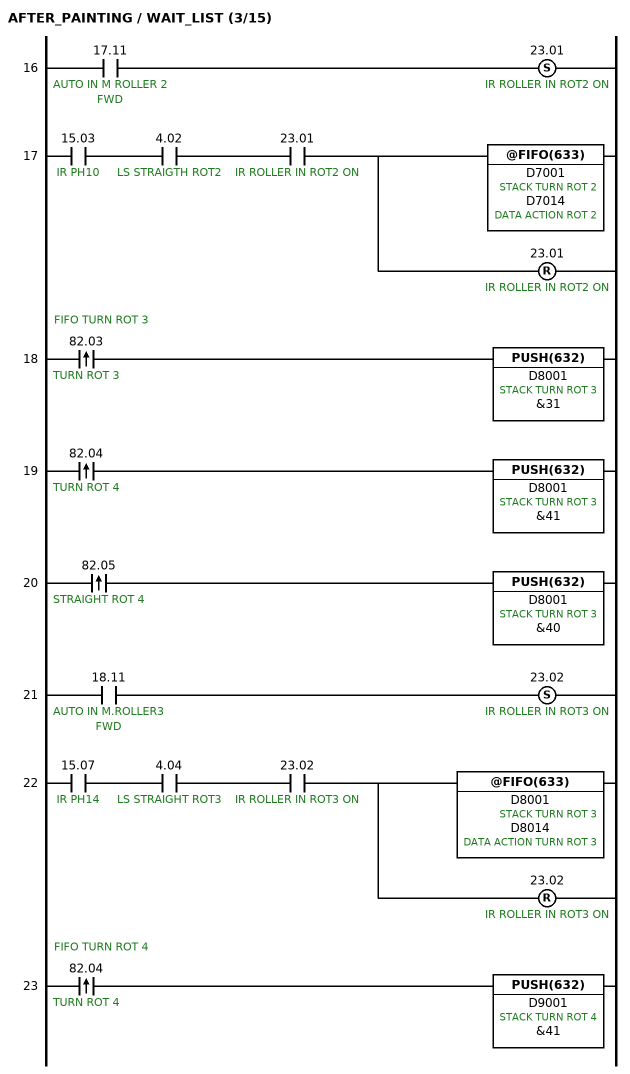
; rung 16
LD 17.11  ; AUTO IN M ROLLER 2 FWD
SET 23.01  ; IR ROLLER IN ROT2 ON
; rung 17
LD 15.03  ; IR PH10
AND 4.02  ; LS STRAIGTH ROT2
AND 23.01  ; IR ROLLER IN ROT2 ON
@FIFO(633) D7001 D7014  ; STACK TURN ROT 2, DATA ACTION ROT 2
RSET 23.01  ; IR ROLLER IN ROT2 ON
; rung 18: FIFO TURN ROT 3
@LD 82.03  ; TURN ROT 3
PUSH(632) D8001 &31  ; STACK TURN ROT 3
; rung 19
@LD 82.04  ; TURN ROT 4
PUSH(632) D8001 &41  ; STACK TURN ROT 3
; rung 20
@LD 82.05  ; STRAIGHT ROT 4
PUSH(632) D8001 &40  ; STACK TURN ROT 3
; rung 21
LD 18.11  ; AUTO IN M.ROLLER3 FWD
SET 23.02  ; IR ROLLER IN ROT3 ON
; rung 22
LD 15.07  ; IR PH14
AND 4.04  ; LS STRAIGHT ROT3
AND 23.02  ; IR ROLLER IN ROT3 ON
@FIFO(633) D8001 D8014  ; STACK TURN ROT 3, DATA ACTION TURN ROT 3
RSET 23.02  ; IR ROLLER IN ROT3 ON
; rung 23: FIFO TURN ROT 4
@LD 82.04  ; TURN ROT 4
PUSH(632) D9001 &41  ; STACK TURN ROT 4

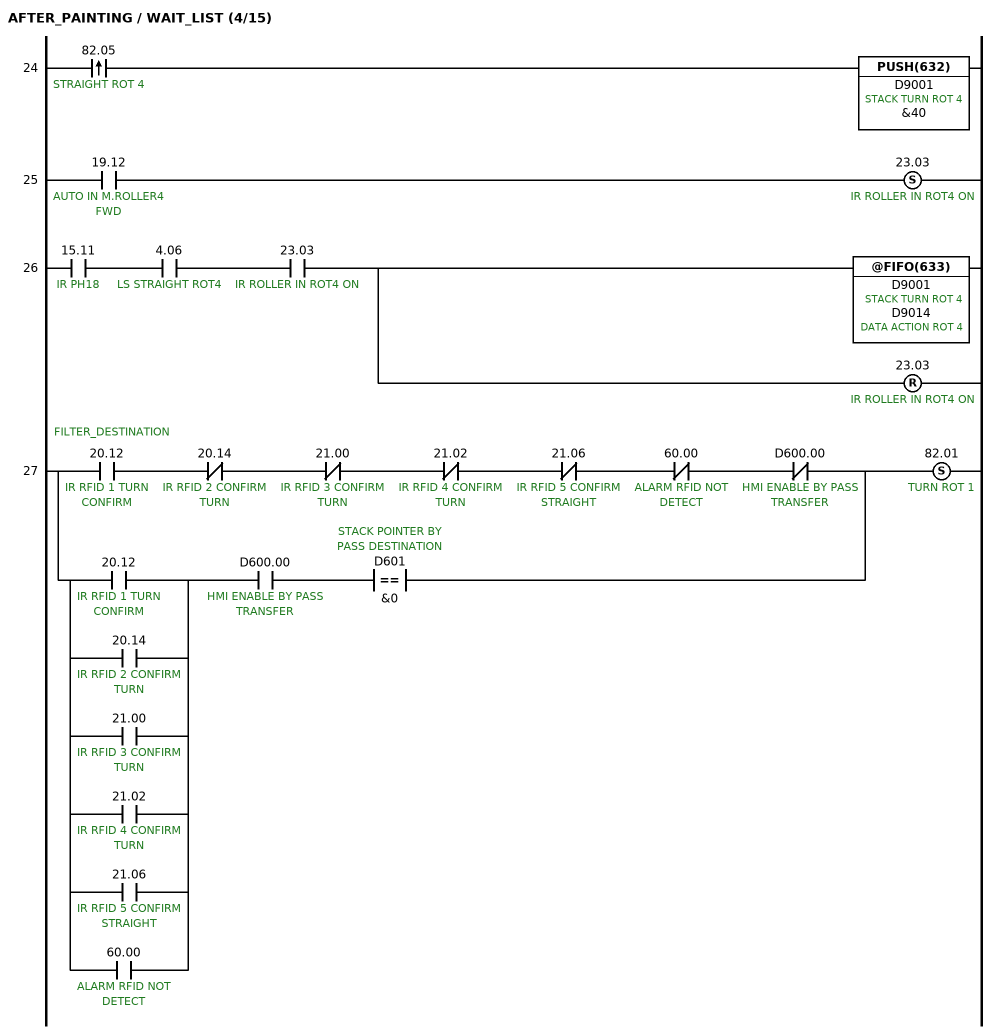
; rung 24
@LD 82.05  ; STRAIGHT ROT 4
PUSH(632) D9001 &40  ; STACK TURN ROT 4
; rung 25
LD 19.12  ; AUTO IN M.ROLLER4 FWD
SET 23.03  ; IR ROLLER IN ROT4 ON
; rung 26
LD 15.11  ; IR PH18
AND 4.06  ; LS STRAIGHT ROT4
AND 23.03  ; IR ROLLER IN ROT4 ON
@FIFO(633) D9001 D9014  ; STACK TURN ROT 4, DATA ACTION ROT 4
RSET 23.03  ; IR ROLLER IN ROT4 ON
; rung 27: FILTER_DESTINATION
LD 20.12  ; IR RFID 1 TURN CONFIRM
ANDNOT 20.14  ; IR RFID 2 CONFIRM TURN
ANDNOT 21.00  ; IR RFID 3 CONFIRM TURN
ANDNOT 21.02  ; IR RFID 4 CONFIRM TURN
ANDNOT 21.06  ; IR RFID 5 CONFIRM STRAIGHT
ANDNOT 60.00  ; ALARM RFID NOT DETECT
ANDNOT D600.00  ; HMI ENABLE BY PASS TRANSFER
LD 20.12  ; IR RFID 1 TURN CONFIRM
OR 20.14  ; IR RFID 2 CONFIRM TURN
OR 21.00  ; IR RFID 3 CONFIRM TURN
OR 21.02  ; IR RFID 4 CONFIRM TURN
OR 21.06  ; IR RFID 5 CONFIRM STRAIGHT
OR 60.00  ; ALARM RFID NOT DETECT
AND D600.00  ; HMI ENABLE BY PASS TRANSFER
AND=(300) D601 &0  ; STACK POINTER BY PASS DESTINATION
ORLD
SET 82.01  ; TURN ROT 1

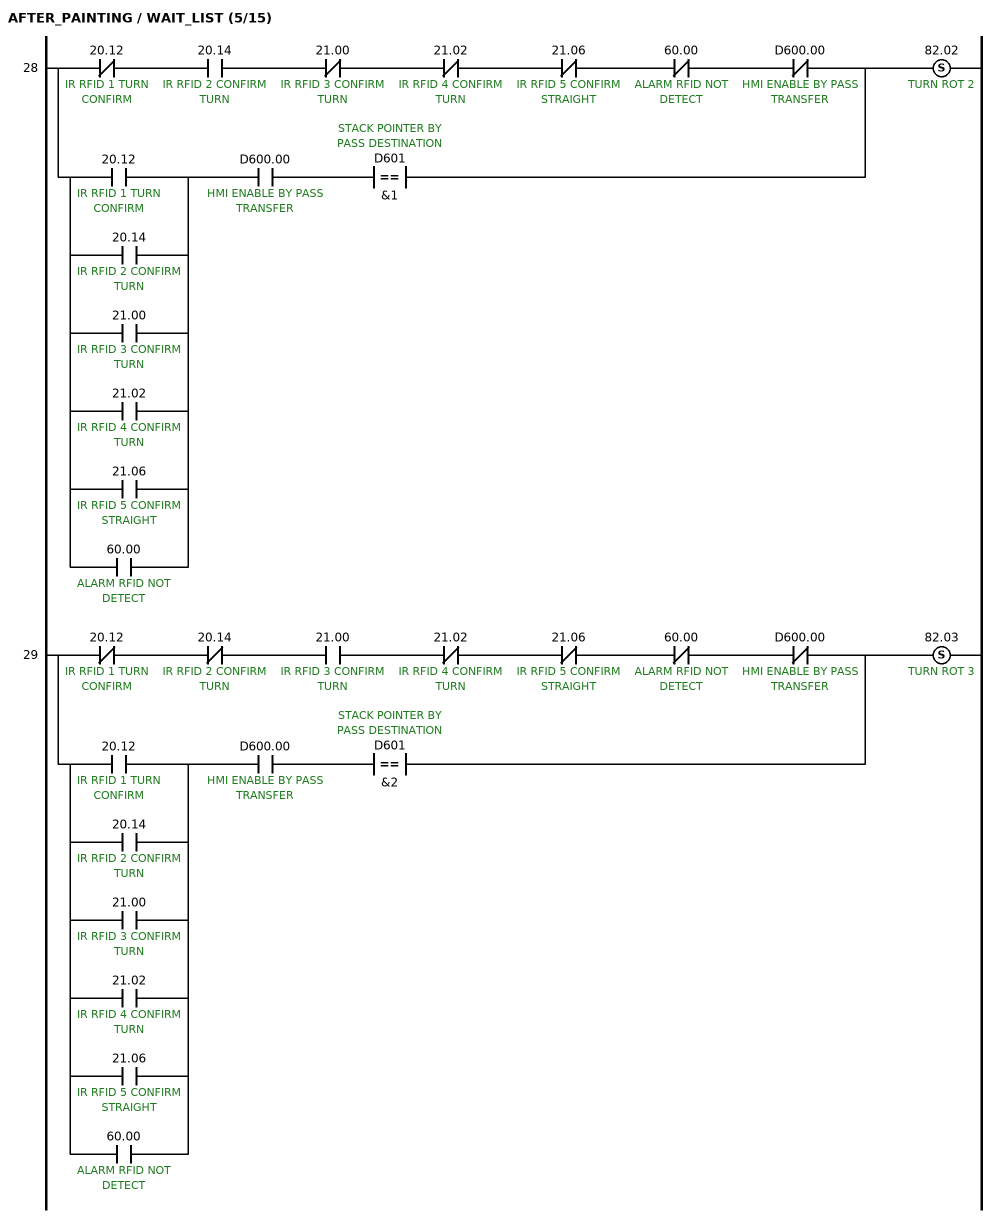
; rung 28
LDNOT 20.12  ; IR RFID 1 TURN CONFIRM
AND 20.14  ; IR RFID 2 CONFIRM TURN
ANDNOT 21.00  ; IR RFID 3 CONFIRM TURN
ANDNOT 21.02  ; IR RFID 4 CONFIRM TURN
ANDNOT 21.06  ; IR RFID 5 CONFIRM STRAIGHT
ANDNOT 60.00  ; ALARM RFID NOT DETECT
ANDNOT D600.00  ; HMI ENABLE BY PASS TRANSFER
LD 20.12  ; IR RFID 1 TURN CONFIRM
OR 20.14  ; IR RFID 2 CONFIRM TURN
OR 21.00  ; IR RFID 3 CONFIRM TURN
OR 21.02  ; IR RFID 4 CONFIRM TURN
OR 21.06  ; IR RFID 5 CONFIRM STRAIGHT
OR 60.00  ; ALARM RFID NOT DETECT
AND D600.00  ; HMI ENABLE BY PASS TRANSFER
AND=(300) D601 &1  ; STACK POINTER BY PASS DESTINATION
ORLD
SET 82.02  ; TURN ROT 2
; rung 29
LDNOT 20.12  ; IR RFID 1 TURN CONFIRM
ANDNOT 20.14  ; IR RFID 2 CONFIRM TURN
AND 21.00  ; IR RFID 3 CONFIRM TURN
ANDNOT 21.02  ; IR RFID 4 CONFIRM TURN
ANDNOT 21.06  ; IR RFID 5 CONFIRM STRAIGHT
ANDNOT 60.00  ; ALARM RFID NOT DETECT
ANDNOT D600.00  ; HMI ENABLE BY PASS TRANSFER
LD 20.12  ; IR RFID 1 TURN CONFIRM
OR 20.14  ; IR RFID 2 CONFIRM TURN
OR 21.00  ; IR RFID 3 CONFIRM TURN
OR 21.02  ; IR RFID 4 CONFIRM TURN
OR 21.06  ; IR RFID 5 CONFIRM STRAIGHT
OR 60.00  ; ALARM RFID NOT DETECT
AND D600.00  ; HMI ENABLE BY PASS TRANSFER
AND=(300) D601 &2  ; STACK POINTER BY PASS DESTINATION
ORLD
SET 82.03  ; TURN ROT 3

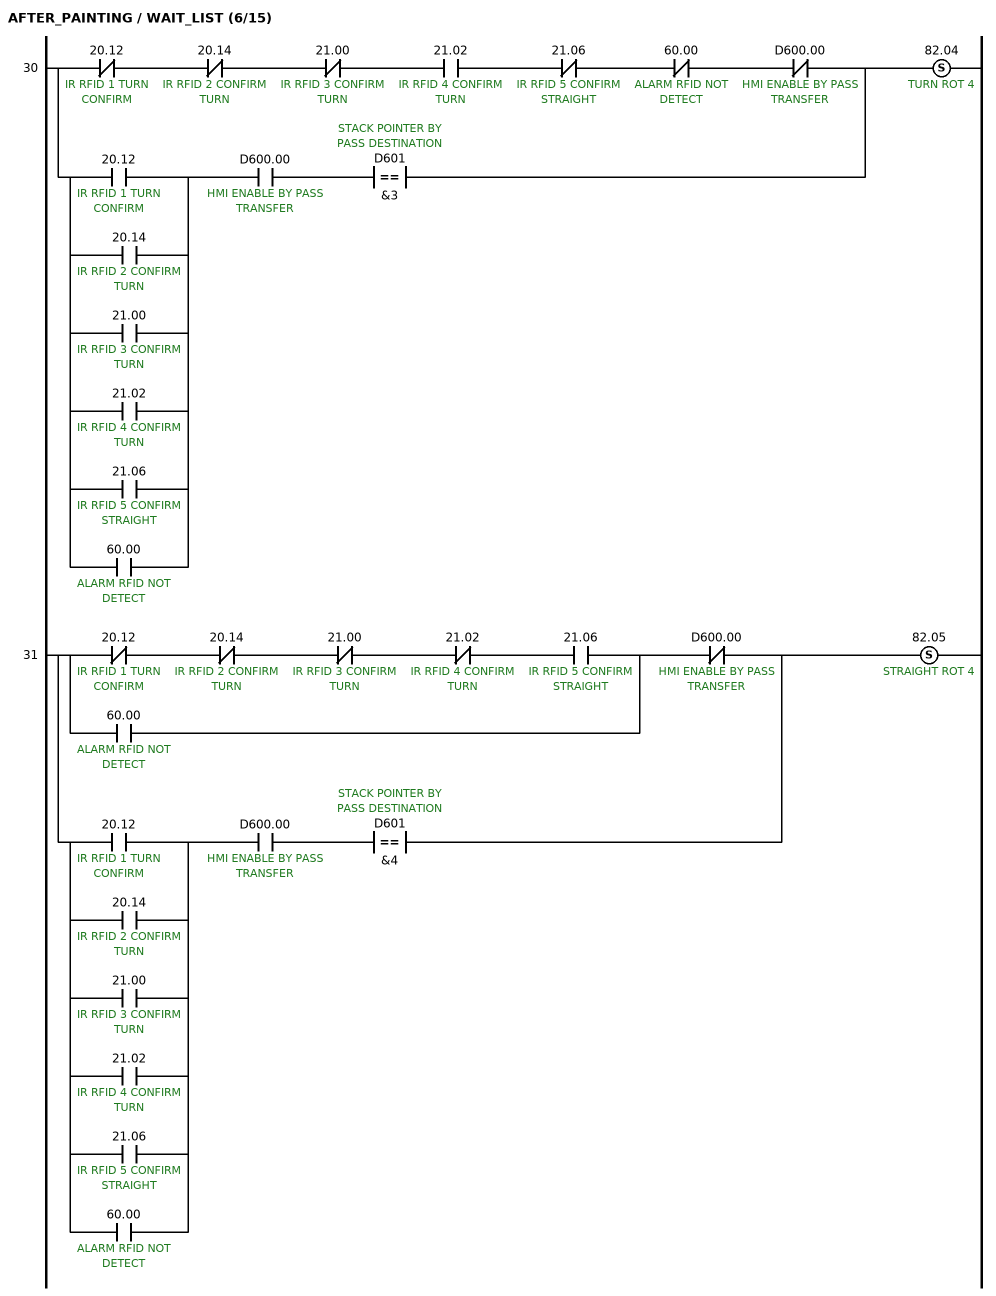
; rung 30
LDNOT 20.12  ; IR RFID 1 TURN CONFIRM
ANDNOT 20.14  ; IR RFID 2 CONFIRM TURN
ANDNOT 21.00  ; IR RFID 3 CONFIRM TURN
AND 21.02  ; IR RFID 4 CONFIRM TURN
ANDNOT 21.06  ; IR RFID 5 CONFIRM STRAIGHT
ANDNOT 60.00  ; ALARM RFID NOT DETECT
ANDNOT D600.00  ; HMI ENABLE BY PASS TRANSFER
LD 20.12  ; IR RFID 1 TURN CONFIRM
OR 20.14  ; IR RFID 2 CONFIRM TURN
OR 21.00  ; IR RFID 3 CONFIRM TURN
OR 21.02  ; IR RFID 4 CONFIRM TURN
OR 21.06  ; IR RFID 5 CONFIRM STRAIGHT
OR 60.00  ; ALARM RFID NOT DETECT
AND D600.00  ; HMI ENABLE BY PASS TRANSFER
AND=(300) D601 &3  ; STACK POINTER BY PASS DESTINATION
ORLD
SET 82.04  ; TURN ROT 4
; rung 31
LDNOT 20.12  ; IR RFID 1 TURN CONFIRM
ANDNOT 20.14  ; IR RFID 2 CONFIRM TURN
ANDNOT 21.00  ; IR RFID 3 CONFIRM TURN
ANDNOT 21.02  ; IR RFID 4 CONFIRM TURN
AND 21.06  ; IR RFID 5 CONFIRM STRAIGHT
OR 60.00  ; ALARM RFID NOT DETECT
ANDNOT D600.00  ; HMI ENABLE BY PASS TRANSFER
LD 20.12  ; IR RFID 1 TURN CONFIRM
OR 20.14  ; IR RFID 2 CONFIRM TURN
OR 21.00  ; IR RFID 3 CONFIRM TURN
OR 21.02  ; IR RFID 4 CONFIRM TURN
OR 21.06  ; IR RFID 5 CONFIRM STRAIGHT
OR 60.00  ; ALARM RFID NOT DETECT
AND D600.00  ; HMI ENABLE BY PASS TRANSFER
AND=(300) D601 &4  ; STACK POINTER BY PASS DESTINATION
ORLD
SET 82.05  ; STRAIGHT ROT 4

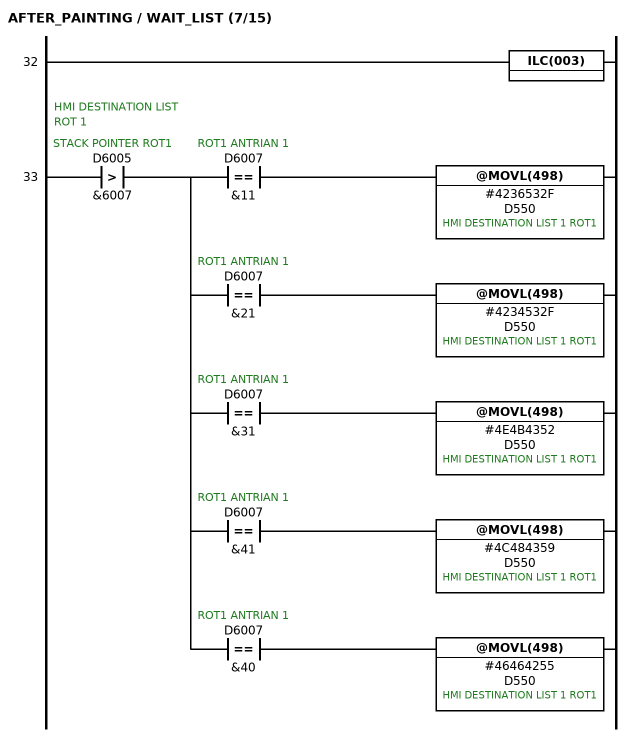
; rung 32
ILC(003)
; rung 33: HMI DESTINATION LIST / ROT 1
LD>(320) D6005 &6007  ; STACK POINTER ROT1
OUT TR0
AND=(300) D6007 &11  ; ROT1 ANTRIAN 1
@MOVL(498) #4236532F D550  ; HMI DESTINATION LIST 1 ROT1
LD TR0
AND=(300) D6007 &21  ; ROT1 ANTRIAN 1
@MOVL(498) #4234532F D550  ; HMI DESTINATION LIST 1 ROT1
LD TR0
AND=(300) D6007 &31  ; ROT1 ANTRIAN 1
@MOVL(498) #4E4B4352 D550  ; HMI DESTINATION LIST 1 ROT1
LD TR0
AND=(300) D6007 &41  ; ROT1 ANTRIAN 1
@MOVL(498) #4C484359 D550  ; HMI DESTINATION LIST 1 ROT1
LD TR0
AND=(300) D6007 &40  ; ROT1 ANTRIAN 1
@MOVL(498) #46464255 D550  ; HMI DESTINATION LIST 1 ROT1

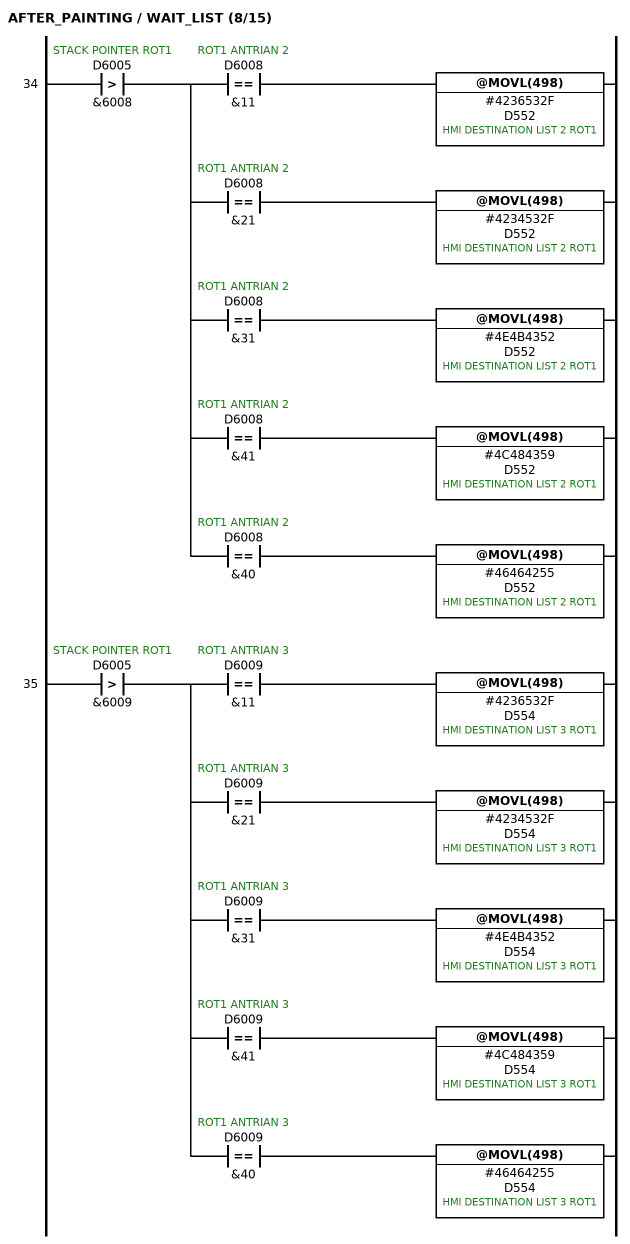
; rung 34
LD>(320) D6005 &6008  ; STACK POINTER ROT1
OUT TR0
AND=(300) D6008 &11  ; ROT1 ANTRIAN 2
@MOVL(498) #4236532F D552  ; HMI DESTINATION LIST 2 ROT1
LD TR0
AND=(300) D6008 &21  ; ROT1 ANTRIAN 2
@MOVL(498) #4234532F D552  ; HMI DESTINATION LIST 2 ROT1
LD TR0
AND=(300) D6008 &31  ; ROT1 ANTRIAN 2
@MOVL(498) #4E4B4352 D552  ; HMI DESTINATION LIST 2 ROT1
LD TR0
AND=(300) D6008 &41  ; ROT1 ANTRIAN 2
@MOVL(498) #4C484359 D552  ; HMI DESTINATION LIST 2 ROT1
LD TR0
AND=(300) D6008 &40  ; ROT1 ANTRIAN 2
@MOVL(498) #46464255 D552  ; HMI DESTINATION LIST 2 ROT1
; rung 35
LD>(320) D6005 &6009  ; STACK POINTER ROT1
OUT TR0
AND=(300) D6009 &11  ; ROT1 ANTRIAN 3
@MOVL(498) #4236532F D554  ; HMI DESTINATION LIST 3 ROT1
LD TR0
AND=(300) D6009 &21  ; ROT1 ANTRIAN 3
@MOVL(498) #4234532F D554  ; HMI DESTINATION LIST 3 ROT1
LD TR0
AND=(300) D6009 &31  ; ROT1 ANTRIAN 3
@MOVL(498) #4E4B4352 D554  ; HMI DESTINATION LIST 3 ROT1
LD TR0
AND=(300) D6009 &41  ; ROT1 ANTRIAN 3
@MOVL(498) #4C484359 D554  ; HMI DESTINATION LIST 3 ROT1
LD TR0
AND=(300) D6009 &40  ; ROT1 ANTRIAN 3
@MOVL(498) #46464255 D554  ; HMI DESTINATION LIST 3 ROT1

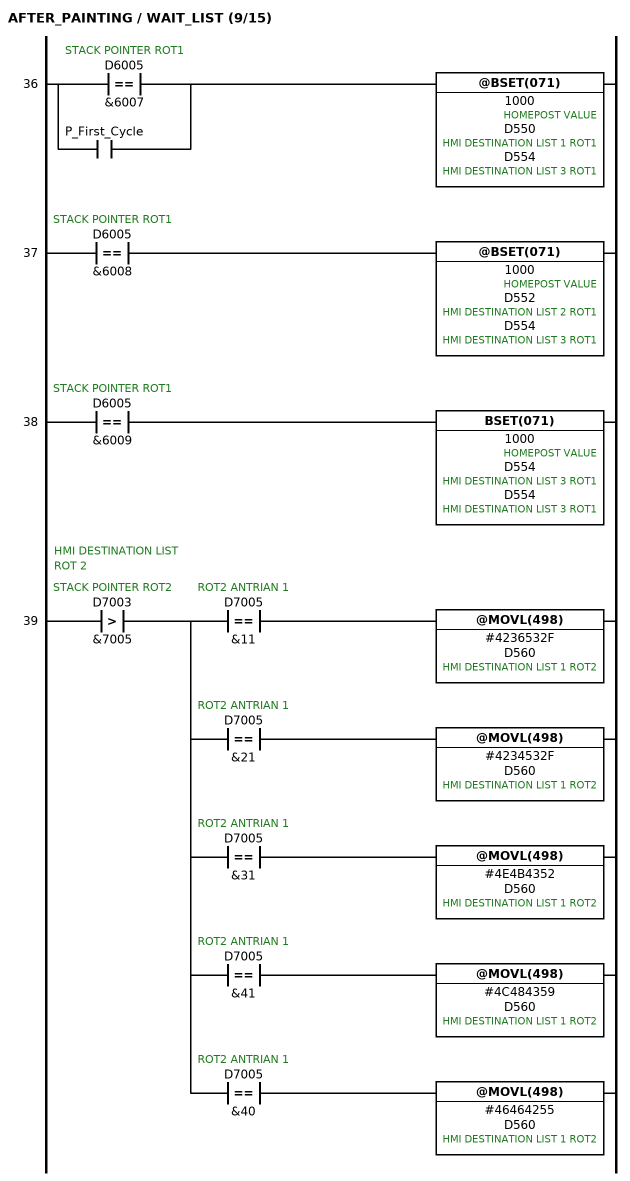
; rung 36
LD=(300) D6005 &6007  ; STACK POINTER ROT1
OR P_First_Cycle
@BSET(071) 1000 D550 D554  ; HOMEPOST VALUE, HMI DESTINATION LIST 1 ROT1, HMI DESTINATION LIST 3 ROT1
; rung 37
LD=(300) D6005 &6008  ; STACK POINTER ROT1
@BSET(071) 1000 D552 D554  ; HOMEPOST VALUE, HMI DESTINATION LIST 2 ROT1, HMI DESTINATION LIST 3 ROT1
; rung 38
LD=(300) D6005 &6009  ; STACK POINTER ROT1
BSET(071) 1000 D554 D554  ; HOMEPOST VALUE, HMI DESTINATION LIST 3 ROT1
; rung 39: HMI DESTINATION LIST / ROT 2
LD>(320) D7003 &7005  ; STACK POINTER ROT2
OUT TR0
AND=(300) D7005 &11  ; ROT2 ANTRIAN 1
@MOVL(498) #4236532F D560  ; HMI DESTINATION LIST 1 ROT2
LD TR0
AND=(300) D7005 &21  ; ROT2 ANTRIAN 1
@MOVL(498) #4234532F D560  ; HMI DESTINATION LIST 1 ROT2
LD TR0
AND=(300) D7005 &31  ; ROT2 ANTRIAN 1
@MOVL(498) #4E4B4352 D560  ; HMI DESTINATION LIST 1 ROT2
LD TR0
AND=(300) D7005 &41  ; ROT2 ANTRIAN 1
@MOVL(498) #4C484359 D560  ; HMI DESTINATION LIST 1 ROT2
LD TR0
AND=(300) D7005 &40  ; ROT2 ANTRIAN 1
@MOVL(498) #46464255 D560  ; HMI DESTINATION LIST 1 ROT2

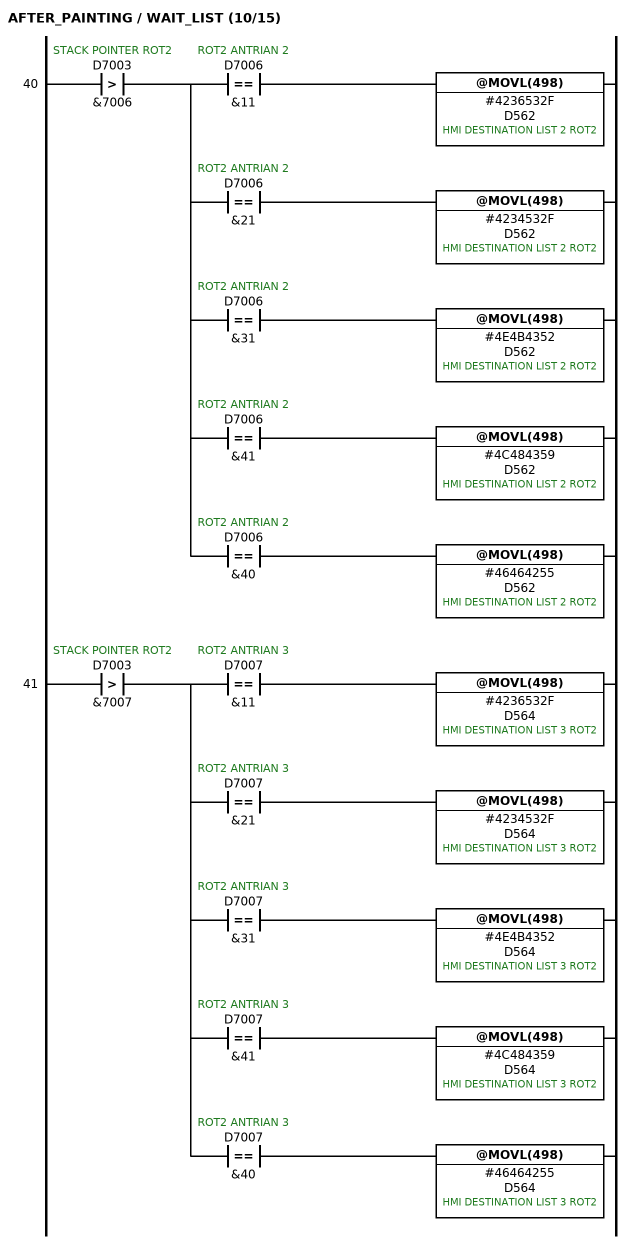
; rung 40
LD>(320) D7003 &7006  ; STACK POINTER ROT2
OUT TR0
AND=(300) D7006 &11  ; ROT2 ANTRIAN 2
@MOVL(498) #4236532F D562  ; HMI DESTINATION LIST 2 ROT2
LD TR0
AND=(300) D7006 &21  ; ROT2 ANTRIAN 2
@MOVL(498) #4234532F D562  ; HMI DESTINATION LIST 2 ROT2
LD TR0
AND=(300) D7006 &31  ; ROT2 ANTRIAN 2
@MOVL(498) #4E4B4352 D562  ; HMI DESTINATION LIST 2 ROT2
LD TR0
AND=(300) D7006 &41  ; ROT2 ANTRIAN 2
@MOVL(498) #4C484359 D562  ; HMI DESTINATION LIST 2 ROT2
LD TR0
AND=(300) D7006 &40  ; ROT2 ANTRIAN 2
@MOVL(498) #46464255 D562  ; HMI DESTINATION LIST 2 ROT2
; rung 41
LD>(320) D7003 &7007  ; STACK POINTER ROT2
OUT TR0
AND=(300) D7007 &11  ; ROT2 ANTRIAN 3
@MOVL(498) #4236532F D564  ; HMI DESTINATION LIST 3 ROT2
LD TR0
AND=(300) D7007 &21  ; ROT2 ANTRIAN 3
@MOVL(498) #4234532F D564  ; HMI DESTINATION LIST 3 ROT2
LD TR0
AND=(300) D7007 &31  ; ROT2 ANTRIAN 3
@MOVL(498) #4E4B4352 D564  ; HMI DESTINATION LIST 3 ROT2
LD TR0
AND=(300) D7007 &41  ; ROT2 ANTRIAN 3
@MOVL(498) #4C484359 D564  ; HMI DESTINATION LIST 3 ROT2
LD TR0
AND=(300) D7007 &40  ; ROT2 ANTRIAN 3
@MOVL(498) #46464255 D564  ; HMI DESTINATION LIST 3 ROT2

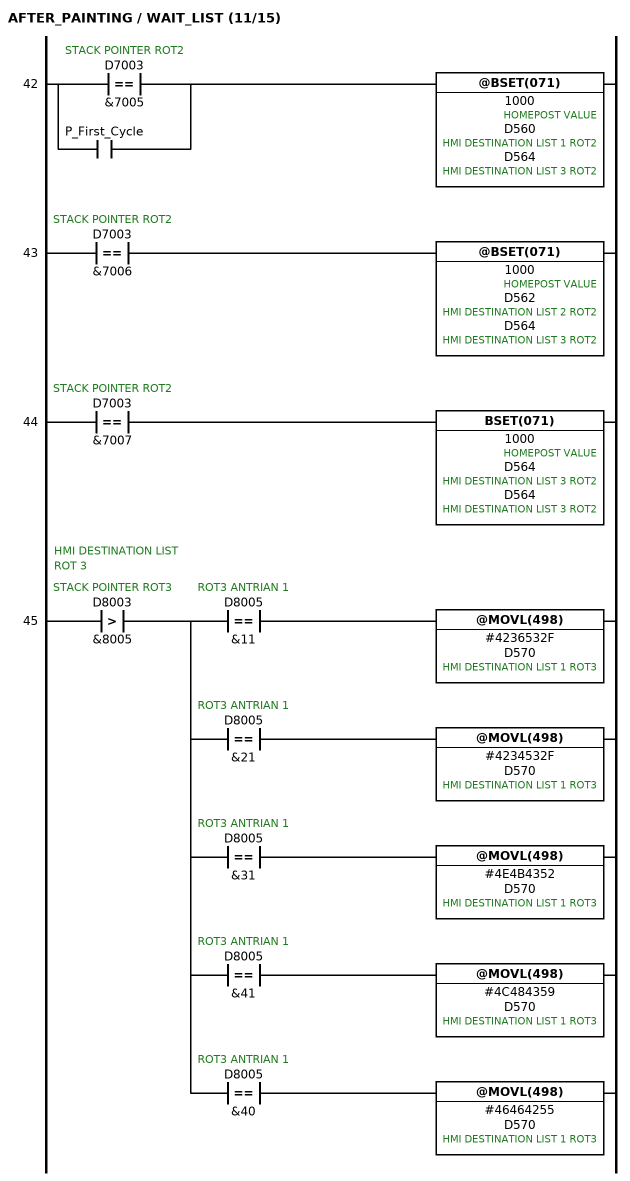
; rung 42
LD=(300) D7003 &7005  ; STACK POINTER ROT2
OR P_First_Cycle
@BSET(071) 1000 D560 D564  ; HOMEPOST VALUE, HMI DESTINATION LIST 1 ROT2, HMI DESTINATION LIST 3 ROT2
; rung 43
LD=(300) D7003 &7006  ; STACK POINTER ROT2
@BSET(071) 1000 D562 D564  ; HOMEPOST VALUE, HMI DESTINATION LIST 2 ROT2, HMI DESTINATION LIST 3 ROT2
; rung 44
LD=(300) D7003 &7007  ; STACK POINTER ROT2
BSET(071) 1000 D564 D564  ; HOMEPOST VALUE, HMI DESTINATION LIST 3 ROT2
; rung 45: HMI DESTINATION LIST / ROT 3
LD>(320) D8003 &8005  ; STACK POINTER ROT3
OUT TR0
AND=(300) D8005 &11  ; ROT3 ANTRIAN 1
@MOVL(498) #4236532F D570  ; HMI DESTINATION LIST 1 ROT3
LD TR0
AND=(300) D8005 &21  ; ROT3 ANTRIAN 1
@MOVL(498) #4234532F D570  ; HMI DESTINATION LIST 1 ROT3
LD TR0
AND=(300) D8005 &31  ; ROT3 ANTRIAN 1
@MOVL(498) #4E4B4352 D570  ; HMI DESTINATION LIST 1 ROT3
LD TR0
AND=(300) D8005 &41  ; ROT3 ANTRIAN 1
@MOVL(498) #4C484359 D570  ; HMI DESTINATION LIST 1 ROT3
LD TR0
AND=(300) D8005 &40  ; ROT3 ANTRIAN 1
@MOVL(498) #46464255 D570  ; HMI DESTINATION LIST 1 ROT3

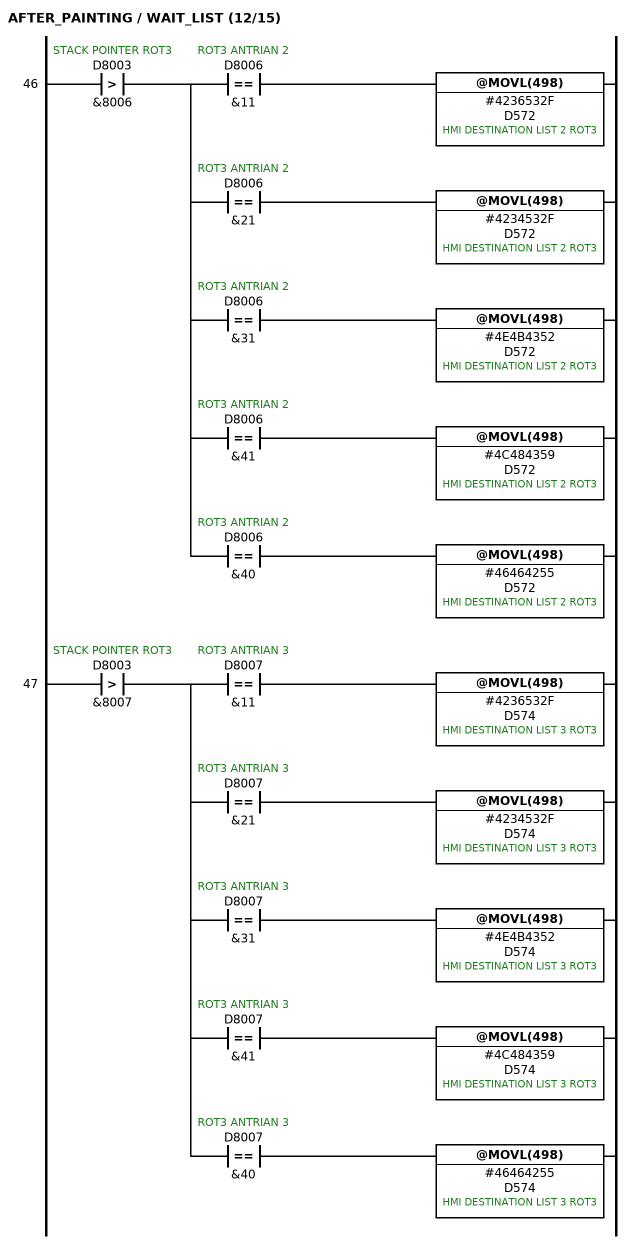
; rung 46
LD>(320) D8003 &8006  ; STACK POINTER ROT3
OUT TR0
AND=(300) D8006 &11  ; ROT3 ANTRIAN 2
@MOVL(498) #4236532F D572  ; HMI DESTINATION LIST 2 ROT3
LD TR0
AND=(300) D8006 &21  ; ROT3 ANTRIAN 2
@MOVL(498) #4234532F D572  ; HMI DESTINATION LIST 2 ROT3
LD TR0
AND=(300) D8006 &31  ; ROT3 ANTRIAN 2
@MOVL(498) #4E4B4352 D572  ; HMI DESTINATION LIST 2 ROT3
LD TR0
AND=(300) D8006 &41  ; ROT3 ANTRIAN 2
@MOVL(498) #4C484359 D572  ; HMI DESTINATION LIST 2 ROT3
LD TR0
AND=(300) D8006 &40  ; ROT3 ANTRIAN 2
@MOVL(498) #46464255 D572  ; HMI DESTINATION LIST 2 ROT3
; rung 47
LD>(320) D8003 &8007  ; STACK POINTER ROT3
OUT TR0
AND=(300) D8007 &11  ; ROT3 ANTRIAN 3
@MOVL(498) #4236532F D574  ; HMI DESTINATION LIST 3 ROT3
LD TR0
AND=(300) D8007 &21  ; ROT3 ANTRIAN 3
@MOVL(498) #4234532F D574  ; HMI DESTINATION LIST 3 ROT3
LD TR0
AND=(300) D8007 &31  ; ROT3 ANTRIAN 3
@MOVL(498) #4E4B4352 D574  ; HMI DESTINATION LIST 3 ROT3
LD TR0
AND=(300) D8007 &41  ; ROT3 ANTRIAN 3
@MOVL(498) #4C484359 D574  ; HMI DESTINATION LIST 3 ROT3
LD TR0
AND=(300) D8007 &40  ; ROT3 ANTRIAN 3
@MOVL(498) #46464255 D574  ; HMI DESTINATION LIST 3 ROT3

